legal notes
=================
| SPDX-FileCopyrightText: © 2022 ekvip automation GmbH <info@ekvip.de>
| SPDX-License-Identifier: Apache-2.0
| For details check: Apache-2.0_

.. _Apache-2.0: https://www.apache.org/licenses/LICENSE-2.0

.. _Apache-2.THIS^.SIZE_ZERO: https://www.apache.org/licenses/LICENSE-2.THIS^.SIZE_ZERO

.. </legal notes>

*)

METHOD runMemoryAreaIsNotDynamicTests
VAR
	foo				:__XWORD;
	stackAddress	:PVOID;
END_VAR
RETURN (NOT TcUnit.TEST_ORDERED(THIS^.getTestNameFor('memoryAreaIsNotDynamic')));
stackAddress := ADR(foo);

THIS^.testMemoryAreaIsNotDynamic(
	address := THIS,
	sizeInBytes := THIS^.I_AM_FAT,
	symbol := 'THIS'
);
THIS^.testMemoryAreaIsNotDynamic(
	address := THIS^.NULL_POINTER,
	sizeInBytes := THIS^.SIZE_ZERO,
	symbol := 'THIS^.NULL_POINTER'
);
THIS^.testMemoryAreaIsNotDynamic(
	address := stackAddress,
	sizeInBytes := SIZEOF(__XWORD),
	symbol := 'stackAddress'
);
THIS^.testMemoryAreaIsNotDynamic(
	address := THIS^.oneByte,
	sizeInBytes := SIZEOF(BYTE),
	symbol := 'THIS^.oneByte'
);
THIS^.testMemoryAreaIsNotDynamic(
	address := THIS^.byteArray,
	sizeInBytes := THIS^.ARRAY_SIZE,
	symbol := 'THIS^.byteArray'
);
THIS^.testMemoryAreaIsNotDynamic(
	address := THIS^.cncAddress,
	sizeInBytes := THIS^.cncSize,
	symbol := 'THIS^.cncAddress'
);
THIS^.testMemoryAreaIsNotDynamic(
	address := THIS^.itsMeAgain,
	sizeInBytes := SIZEOF(PVOID),
	symbol := 'THIS^.itsMeAgain'
);
THIS^.testMemoryAreaIsNotDynamic(
	address := THIS^.itsMeAgain^,
	sizeInBytes := THIS^.I_AM_FAT,
	symbol := 'THIS^.itsMeAgain^'
);
THIS^.testMemoryAreaIsNotDynamic(
	address := THIS^.me,
	sizeInBytes := THIS^.I_AM_FAT,
	symbol := 'THIS^.me'
);
THIS^.testMemoryAreaIsNotDynamic(
	address := THIS^.myMom,
	sizeInBytes := SIZEOF(AbstractAssertorTest),
	symbol := 'THIS^.myMom'
);
THIS^.testMemoryAreaIsNotDynamic(
	address := THIS^.invalidByte,
	sizeInBytes := SIZEOF(BYTE),
	symbol := 'THIS^.invalidByte'
);

THIS^.testMemoryAreaIsNotDynamic(
	address := THIS^.itsMeAgain,
	sizeInBytes := THIS^.SIZE_ZERO,
	symbol := 'THIS^.itsMeAgain'
);
THIS^.testMemoryAreaIsNotDynamic(
	address := THIS,
	sizeInBytes := THIS^.SIZE_ZERO,
	symbol := 'THIS'
);
THIS^.testMemoryAreaIsNotDynamic(
	address := THIS^.NULL_POINTER,
	sizeInBytes := SIZEOF(PVOID),
	symbol := 'THIS^.NULL_POINTER'
);
THIS^.testMemoryAreaIsNotDynamic(
	address := stackAddress,
	sizeInBytes := THIS^.SIZE_ZERO,
	symbol := 'stackAddress'
);
THIS^.testMemoryAreaIsNotDynamic(
	address := THIS^.oneByte,
	sizeInBytes := THIS^.SIZE_ZERO,
	symbol := 'THIS^.oneByte'
);
THIS^.testMemoryAreaIsNotDynamic(
	address := THIS^.byteArray,
	sizeInBytes := THIS^.SIZE_ZERO,
	symbol := 'THIS^.byteArray'
);
THIS^.testMemoryAreaIsNotDynamic(
	address := THIS^.itsMeAgain,
	sizeInBytes := THIS^.SIZE_ZERO,
	symbol := 'THIS^.itsMeAgain'
);
THIS^.testMemoryAreaIsNotDynamic(
	address := THIS^.cncAddress,
	sizeInBytes := THIS^.SIZE_ZERO,
	symbol := 'THIS^.cncAddress'
);
THIS^.testMemoryAreaIsNotDynamic(
	address := THIS^.itsMeAgain^,
	sizeInBytes := THIS^.SIZE_ZERO,
	symbol := 'THIS^.itsMeAgain^'
);
THIS^.testMemoryAreaIsNotDynamic(
	address := THIS^.INVALID_POINTER,
	sizeInBytes := SIZEOF(PVOID),
	symbol := 'THIS^.INVALID_POINTER'
);
THIS^.testMemoryAreaIsNotDynamic(
	address := THIS^.myMom,
	sizeInBytes := THIS^.SIZE_ZERO,
	symbol := 'THIS^.myMom'
);
THIS^.testMemoryAreaIsNotDynamic(
	address := THIS^.invalidByte,
	sizeInBytes := THIS^.SIZE_ZERO,
	symbol := 'THIS^.invalidByte'
);

TcUnit.TEST_FINISHED();
END_METHOD

(*

short summary
==================
This test method tests ``assert.pointers.memoryAreaIsNotStatic``
method of CNM_AssertionInterfaceLib library with various inputs

.. <legal notes>

legal notes
=================
| SPDX-FileCopyrightText: © 2022 ekvip automation GmbH <info@ekvip.de>
| SPDX-License-Identifier: Apache-2.0
| For details check: Apache-2.0_

.. _Apache-2.0: https://www.apache.org/licenses/LICENSE-2.0

.. _Apache-2.THIS^.SIZE_ZERO: https://www.apache.org/licenses/LICENSE-2.THIS^.SIZE_ZERO

.. </legal notes>

*)

METHOD runMemoryAreaIsNotStaticTests
VAR
	foo				:__XWORD;
	stackAddress	:PVOID;
END_VAR
RETURN (NOT TcUnit.TEST_ORDERED(THIS^.getTestNameFor('memoryAreaIsNotStatic')));
stackAddress := ADR(foo);

THIS^.testMemoryAreaIsNotStatic(
	address := THIS,
	sizeInBytes := THIS^.I_AM_FAT,
	symbol := 'THIS'
);
THIS^.testMemoryAreaIsNotStatic(
	address := THIS^.NULL_POINTER,
	sizeInBytes := THIS^.SIZE_ZERO,
	symbol := 'THIS^.NULL_POINTER'
);
THIS^.testMemoryAreaIsNotStatic(
	address := stackAddress,
	sizeInBytes := SIZEOF(__XWORD),
	symbol := 'stackAddress'
);
THIS^.testMemoryAreaIsNotStatic(
	address := THIS^.oneByte,
	sizeInBytes := SIZEOF(BYTE),
	symbol := 'THIS^.oneByte'
);
THIS^.testMemoryAreaIsNotStatic(
	address := THIS^.byteArray,
	sizeInBytes := THIS^.ARRAY_SIZE,
	symbol := 'THIS^.byteArray'
);
THIS^.testMemoryAreaIsNotStatic(
	address := THIS^.cncAddress,
	sizeInBytes := THIS^.cncSize,
	symbol := 'THIS^.cncAddress'
);
THIS^.testMemoryAreaIsNotStatic(
	address := THIS^.itsMeAgain,
	sizeInBytes := SIZEOF(PVOID),
	symbol := 'THIS^.itsMeAgain'
);
THIS^.testMemoryAreaIsNotStatic(
	address := THIS^.itsMeAgain^,
	sizeInBytes := THIS^.I_AM_FAT,
	symbol := 'THIS^.itsMeAgain^'
);
THIS^.testMemoryAreaIsNotStatic(
	address := THIS^.me,
	sizeInBytes := THIS^.I_AM_FAT,
	symbol := 'THIS^.me'
);
THIS^.testMemoryAreaIsNotStatic(
	address := THIS^.myMom,
	sizeInBytes := SIZEOF(AbstractAssertorTest),
	symbol := 'THIS^.myMom'
);
THIS^.testMemoryAreaIsNotStatic(
	address := THIS^.invalidByte,
	sizeInBytes := SIZEOF(BYTE),
	symbol := 'THIS^.invalidByte'
);

THIS^.testMemoryAreaIsNotStatic(
	address := THIS^.itsMeAgain,
	sizeInBytes := THIS^.SIZE_ZERO,
	symbol := 'THIS^.itsMeAgain'
);
THIS^.testMemoryAreaIsNotStatic(
	address := THIS,
	sizeInBytes := THIS^.SIZE_ZERO,
	symbol := 'THIS'
);
THIS^.testMemoryAreaIsNotStatic(
	address := THIS^.NULL_POINTER,
	sizeInBytes := SIZEOF(PVOID),
	symbol := 'THIS^.NULL_POINTER'
);
THIS^.testMemoryAreaIsNotStatic(
	address := stackAddress,
	sizeInBytes := THIS^.SIZE_ZERO,
	symbol := 'stackAddress'
);
THIS^.testMemoryAreaIsNotStatic(
	address := THIS^.oneByte,
	sizeInBytes := THIS^.SIZE_ZERO,
	symbol := 'THIS^.oneByte'
);
THIS^.testMemoryAreaIsNotStatic(
	address := THIS^.byteArray,
	sizeInBytes := THIS^.SIZE_ZERO,
	symbol := 'THIS^.byteArray'
);
THIS^.testMemoryAreaIsNotStatic(
	address := THIS^.itsMeAgain,
	sizeInBytes := THIS^.SIZE_ZERO,
	symbol := 'THIS^.itsMeAgain'
);
THIS^.testMemoryAreaIsNotStatic(
	address := THIS^.cncAddress,
	sizeInBytes := THIS^.SIZE_ZERO,
	symbol := 'THIS^.cncAddress'
);
THIS^.testMemoryAreaIsNotStatic(
	address := THIS^.itsMeAgain^,
	sizeInBytes := THIS^.SIZE_ZERO,
	symbol := 'THIS^.itsMeAgain^'
);
THIS^.testMemoryAreaIsNotStatic(
	address := THIS^.INVALID_POINTER,
	sizeInBytes := SIZEOF(PVOID),
	symbol := 'THIS^.INVALID_POINTER'
);
THIS^.testMemoryAreaIsNotStatic(
	address := THIS^.myMom,
	sizeInBytes := THIS^.SIZE_ZERO,
	symbol := 'THIS^.myMom'
);
THIS^.testMemoryAreaIsNotStatic(
	address := THIS^.invalidByte,
	sizeInBytes := THIS^.SIZE_ZERO,
	symbol := 'THIS^.invalidByte'
);

TcUnit.TEST_FINISHED();
END_METHOD

(*

short summary
==================
This test method tests ``assert.pointers.memoryAreaIsNotUnkown``
method of CNM_AssertionInterfaceLib library with various inputs

.. <legal notes>

legal notes
=================
| SPDX-FileCopyrightText: © 2022 ekvip automation GmbH <info@ekvip.de>
| SPDX-License-Identifier: Apache-2.0
| For details check: Apache-2.0_

.. _Apache-2.0: https://www.apache.org/licenses/LICENSE-2.0

.. _Apache-2.THIS^.SIZE_ZERO: https://www.apache.org/licenses/LICENSE-2.THIS^.SIZE_ZERO

.. </legal notes>

*)

METHOD runMemoryAreaIsNotUnknownTests
VAR
	foo				:__XWORD;
	stackAddress	:PVOID;
END_VAR
RETURN (NOT TcUnit.TEST_ORDERED(THIS^.getTestNameFor('memoryAreaIsNotUnkown')));
stackAddress := ADR(foo);

THIS^.testMemoryAreaIsNotUnknown(
	address := THIS,
	sizeInBytes := THIS^.I_AM_FAT,
	symbol := 'THIS'
);
THIS^.testMemoryAreaIsNotUnknown(
	address := THIS^.NULL_POINTER,
	sizeInBytes := THIS^.SIZE_ZERO,
	symbol := 'THIS^.NULL_POINTER'
);
THIS^.testMemoryAreaIsNotUnknown(
	address := stackAddress,
	sizeInBytes := SIZEOF(__XWORD),
	symbol := 'stackAddress'
);
THIS^.testMemoryAreaIsNotUnknown(
	address := THIS^.oneByte,
	sizeInBytes := SIZEOF(BYTE),
	symbol := 'THIS^.oneByte'
);
THIS^.testMemoryAreaIsNotUnknown(
	address := THIS^.byteArray,
	sizeInBytes := THIS^.ARRAY_SIZE,
	symbol := 'THIS^.byteArray'
);
THIS^.testMemoryAreaIsNotUnknown(
	address := THIS^.cncAddress,
	sizeInBytes := THIS^.cncSize,
	symbol := 'THIS^.cncAddress'
);
THIS^.testMemoryAreaIsNotUnknown(
	address := THIS^.itsMeAgain,
	sizeInBytes := SIZEOF(PVOID),
	symbol := 'THIS^.itsMeAgain'
);
THIS^.testMemoryAreaIsNotUnknown(
	address := THIS^.itsMeAgain^,
	sizeInBytes := THIS^.I_AM_FAT,
	symbol := 'THIS^.itsMeAgain^'
);
THIS^.testMemoryAreaIsNotUnknown(
	address := THIS^.me,
	sizeInBytes := THIS^.I_AM_FAT,
	symbol := 'THIS^.me'
);
THIS^.testMemoryAreaIsNotUnknown(
	address := THIS^.myMom,
	sizeInBytes := SIZEOF(AbstractAssertorTest),
	symbol := 'THIS^.myMom'
);
THIS^.testMemoryAreaIsNotUnknown(
	address := THIS^.invalidByte,
	sizeInBytes := SIZEOF(BYTE),
	symbol := 'THIS^.invalidByte'
);

THIS^.testMemoryAreaIsNotUnknown(
	address := THIS^.itsMeAgain,
	sizeInBytes := THIS^.SIZE_ZERO,
	symbol := 'THIS^.itsMeAgain'
);
THIS^.testMemoryAreaIsNotUnknown(
	address := THIS,
	sizeInBytes := THIS^.SIZE_ZERO,
	symbol := 'THIS'
);
THIS^.testMemoryAreaIsNotUnknown(
	address := THIS^.NULL_POINTER,
	sizeInBytes := SIZEOF(PVOID),
	symbol := 'THIS^.NULL_POINTER'
);
THIS^.testMemoryAreaIsNotUnknown(
	address := stackAddress,
	sizeInBytes := THIS^.SIZE_ZERO,
	symbol := 'stackAddress'
);
THIS^.testMemoryAreaIsNotUnknown(
	address := THIS^.oneByte,
	sizeInBytes := THIS^.SIZE_ZERO,
	symbol := 'THIS^.oneByte'
);
THIS^.testMemoryAreaIsNotUnknown(
	address := THIS^.byteArray,
	sizeInBytes := THIS^.SIZE_ZERO,
	symbol := 'THIS^.byteArray'
);
THIS^.testMemoryAreaIsNotUnknown(
	address := THIS^.itsMeAgain,
	sizeInBytes := THIS^.SIZE_ZERO,
	symbol := 'THIS^.itsMeAgain'
);
THIS^.testMemoryAreaIsNotUnknown(
	address := THIS^.cncAddress,
	sizeInBytes := THIS^.SIZE_ZERO,
	symbol := 'THIS^.cncAddress'
);
THIS^.testMemoryAreaIsNotUnknown(
	address := THIS^.itsMeAgain^,
	sizeInBytes := THIS^.SIZE_ZERO,
	symbol := 'THIS^.itsMeAgain^'
);
THIS^.testMemoryAreaIsNotUnknown(
	address := THIS^.INVALID_POINTER,
	sizeInBytes := SIZEOF(PVOID),
	symbol := 'THIS^.INVALID_POINTER'
);
THIS^.testMemoryAreaIsNotUnknown(
	address := THIS^.myMom,
	sizeInBytes := THIS^.SIZE_ZERO,
	symbol := 'THIS^.myMom'
);
THIS^.testMemoryAreaIsNotUnknown(
	address := THIS^.invalidByte,
	sizeInBytes := THIS^.SIZE_ZERO,
	symbol := 'THIS^.invalidByte'
);

TcUnit.TEST_FINISHED();
END_METHOD

(*

short summary
==================
This test method tests ``assert.pointers.memoryAreaIsStatic``
method of CNM_AssertionInterfaceLib library with various inputs

.. <legal notes>

legal notes
=================
| SPDX-FileCopyrightText: © 2022 ekvip automation GmbH <info@ekvip.de>
| SPDX-License-Identifier: Apache-2.0
| For details check: Apache-2.0_

.. _Apache-2.0: https://www.apache.org/licenses/LICENSE-2.0

.. _Apache-2.THIS^.SIZE_ZERO: https://www.apache.org/licenses/LICENSE-2.THIS^.SIZE_ZERO

.. </legal notes>

*)

METHOD runMemoryAreaIsStaticTests
VAR
	foo				:__XWORD;
	stackAddress	:PVOID;
END_VAR
RETURN (NOT TcUnit.TEST_ORDERED(THIS^.getTestNameFor('memoryAreaIsStatic')));
stackAddress := ADR(foo);

THIS^.testMemoryAreaIsStatic(
	address := THIS,
	sizeInBytes := THIS^.I_AM_FAT,
	symbol := 'THIS'
);
THIS^.testMemoryAreaIsStatic(
	address := THIS^.NULL_POINTER,
	sizeInBytes := THIS^.SIZE_ZERO,
	symbol := 'THIS^.NULL_POINTER'
);
THIS^.testMemoryAreaIsStatic(
	address := stackAddress,
	sizeInBytes := SIZEOF(__XWORD),
	symbol := 'stackAddress'
);
THIS^.testMemoryAreaIsStatic(
	address := THIS^.oneByte,
	sizeInBytes := SIZEOF(BYTE),
	symbol := 'THIS^.oneByte'
);
THIS^.testMemoryAreaIsStatic(
	address := THIS^.byteArray,
	sizeInBytes := THIS^.ARRAY_SIZE,
	symbol := 'THIS^.byteArray'
);
THIS^.testMemoryAreaIsStatic(
	address := THIS^.cncAddress,
	sizeInBytes := THIS^.cncSize,
	symbol := 'THIS^.cncAddress'
);
THIS^.testMemoryAreaIsStatic(
	address := THIS^.itsMeAgain,
	sizeInBytes := SIZEOF(PVOID),
	symbol := 'THIS^.itsMeAgain'
);
THIS^.testMemoryAreaIsStatic(
	address := THIS^.itsMeAgain^,
	sizeInBytes := THIS^.I_AM_FAT,
	symbol := 'THIS^.itsMeAgain^'
);
THIS^.testMemoryAreaIsStatic(
	address := THIS^.me,
	sizeInBytes := THIS^.I_AM_FAT,
	symbol := 'THIS^.me'
);
THIS^.testMemoryAreaIsStatic(
	address := THIS^.myMom,
	sizeInBytes := SIZEOF(AbstractAssertorTest),
	symbol := 'THIS^.myMom'
);
THIS^.testMemoryAreaIsStatic(
	address := THIS^.invalidByte,
	sizeInBytes := SIZEOF(BYTE),
	symbol := 'THIS^.invalidByte'
);

THIS^.testMemoryAreaIsStatic(
	address := THIS^.itsMeAgain,
	sizeInBytes := THIS^.SIZE_ZERO,
	symbol := 'THIS^.itsMeAgain'
);
THIS^.testMemoryAreaIsStatic(
	address := THIS,
	sizeInBytes := THIS^.SIZE_ZERO,
	symbol := 'THIS'
);
THIS^.testMemoryAreaIsStatic(
	address := THIS^.NULL_POINTER,
	sizeInBytes := SIZEOF(PVOID),
	symbol := 'THIS^.NULL_POINTER'
);
THIS^.testMemoryAreaIsStatic(
	address := stackAddress,
	sizeInBytes := THIS^.SIZE_ZERO,
	symbol := 'stackAddress'
);
THIS^.testMemoryAreaIsStatic(
	address := THIS^.oneByte,
	sizeInBytes := THIS^.SIZE_ZERO,
	symbol := 'THIS^.oneByte'
);
THIS^.testMemoryAreaIsStatic(
	address := THIS^.byteArray,
	sizeInBytes := THIS^.SIZE_ZERO,
	symbol := 'THIS^.byteArray'
);
THIS^.testMemoryAreaIsStatic(
	address := THIS^.itsMeAgain,
	sizeInBytes := THIS^.SIZE_ZERO,
	symbol := 'THIS^.itsMeAgain'
);
THIS^.testMemoryAreaIsStatic(
	address := THIS^.cncAddress,
	sizeInBytes := THIS^.SIZE_ZERO,
	symbol := 'THIS^.cncAddress'
);
THIS^.testMemoryAreaIsStatic(
	address := THIS^.itsMeAgain^,
	sizeInBytes := THIS^.SIZE_ZERO,
	symbol := 'THIS^.itsMeAgain^'
);
THIS^.testMemoryAreaIsStatic(
	address := THIS^.INVALID_POINTER,
	sizeInBytes := SIZEOF(PVOID),
	symbol := 'THIS^.INVALID_POINTER'
);
THIS^.testMemoryAreaIsStatic(
	address := THIS^.myMom,
	sizeInBytes := THIS^.SIZE_ZERO,
	symbol := 'THIS^.myMom'
);
THIS^.testMemoryAreaIsStatic(
	address := THIS^.invalidByte,
	sizeInBytes := THIS^.SIZE_ZERO,
	symbol := 'THIS^.invalidByte'
);

TcUnit.TEST_FINISHED();
END_METHOD

(*

short summary
==================
This test method tests ``assert.pointers.memoryAreaIsUnkown``
method of CNM_AssertionInterfaceLib library with various inputs

.. <legal notes>

legal notes
=================
| SPDX-FileCopyrightText: © 2022 ekvip automation GmbH <info@ekvip.de>
| SPDX-License-Identifier: Apache-2.0
| For details check: Apache-2.0_

.. _Apache-2.0: https://www.apache.org/licenses/LICENSE-2.0

.. _Apache-2.THIS^.SIZE_ZERO: https://www.apache.org/licenses/LICENSE-2.THIS^.SIZE_ZERO

.. </legal notes>

*)

METHOD runMemoryAreaIsUnknownTests
VAR
	foo				:__XWORD;
	stackAddress	:PVOID;
END_VAR
RETURN (NOT TcUnit.TEST_ORDERED(THIS^.getTestNameFor('memoryAreaIsUnkown')));
stackAddress := ADR(foo);

THIS^.testMemoryAreaIsUnknown(
	address := THIS,
	sizeInBytes := THIS^.I_AM_FAT,
	symbol := 'THIS'
);
THIS^.testMemoryAreaIsUnknown(
	address := THIS^.NULL_POINTER,
	sizeInBytes := THIS^.SIZE_ZERO,
	symbol := 'THIS^.NULL_POINTER'
);
THIS^.testMemoryAreaIsUnknown(
	address := stackAddress,
	sizeInBytes := SIZEOF(__XWORD),
	symbol := 'stackAddress'
);
THIS^.testMemoryAreaIsUnknown(
	address := THIS^.oneByte,
	sizeInBytes := SIZEOF(BYTE),
	symbol := 'THIS^.oneByte'
);
THIS^.testMemoryAreaIsUnknown(
	address := THIS^.byteArray,
	sizeInBytes := THIS^.ARRAY_SIZE,
	symbol := 'THIS^.byteArray'
);
THIS^.testMemoryAreaIsUnknown(
	address := THIS^.cncAddress,
	sizeInBytes := THIS^.cncSize,
	symbol := 'THIS^.cncAddress'
);
THIS^.testMemoryAreaIsUnknown(
	address := THIS^.itsMeAgain,
	sizeInBytes := SIZEOF(PVOID),
	symbol := 'THIS^.itsMeAgain'
);
THIS^.testMemoryAreaIsUnknown(
	address := THIS^.itsMeAgain^,
	sizeInBytes := THIS^.I_AM_FAT,
	symbol := 'THIS^.itsMeAgain^'
);
THIS^.testMemoryAreaIsUnknown(
	address := THIS^.me,
	sizeInBytes := THIS^.I_AM_FAT,
	symbol := 'THIS^.me'
);
THIS^.testMemoryAreaIsUnknown(
	address := THIS^.myMom,
	sizeInBytes := SIZEOF(AbstractAssertorTest),
	symbol := 'THIS^.myMom'
);
THIS^.testMemoryAreaIsUnknown(
	address := THIS^.invalidByte,
	sizeInBytes := SIZEOF(BYTE),
	symbol := 'THIS^.invalidByte'
);

THIS^.testMemoryAreaIsUnknown(
	address := THIS^.itsMeAgain,
	sizeInBytes := THIS^.SIZE_ZERO,
	symbol := 'THIS^.itsMeAgain'
);
THIS^.testMemoryAreaIsUnknown(
	address := THIS,
	sizeInBytes := THIS^.SIZE_ZERO,
	symbol := 'THIS'
);
THIS^.testMemoryAreaIsUnknown(
	address := THIS^.NULL_POINTER,
	sizeInBytes := SIZEOF(PVOID),
	symbol := 'THIS^.NULL_POINTER'
);
THIS^.testMemoryAreaIsUnknown(
	address := stackAddress,
	sizeInBytes := THIS^.SIZE_ZERO,
	symbol := 'stackAddress'
);
THIS^.testMemoryAreaIsUnknown(
	address := THIS^.oneByte,
	sizeInBytes := THIS^.SIZE_ZERO,
	symbol := 'THIS^.oneByte'
);
THIS^.testMemoryAreaIsUnknown(
	address := THIS^.byteArray,
	sizeInBytes := THIS^.SIZE_ZERO,
	symbol := 'THIS^.byteArray'
);
THIS^.testMemoryAreaIsUnknown(
	address := THIS^.itsMeAgain,
	sizeInBytes := THIS^.SIZE_ZERO,
	symbol := 'THIS^.itsMeAgain'
);
THIS^.testMemoryAreaIsUnknown(
	address := THIS^.cncAddress,
	sizeInBytes := THIS^.SIZE_ZERO,
	symbol := 'THIS^.cncAddress'
);
THIS^.testMemoryAreaIsUnknown(
	address := THIS^.itsMeAgain^,
	sizeInBytes := THIS^.SIZE_ZERO,
	symbol := 'THIS^.itsMeAgain^'
);
THIS^.testMemoryAreaIsUnknown(
	address := THIS^.INVALID_POINTER,
	sizeInBytes := SIZEOF(PVOID),
	symbol := 'THIS^.INVALID_POINTER'
);
THIS^.testMemoryAreaIsUnknown(
	address := THIS^.myMom,
	sizeInBytes := THIS^.SIZE_ZERO,
	symbol := 'THIS^.myMom'
);
THIS^.testMemoryAreaIsUnknown(
	address := THIS^.invalidByte,
	sizeInBytes := THIS^.SIZE_ZERO,
	symbol := 'THIS^.invalidByte'
);

TcUnit.TEST_FINISHED();
END_METHOD

(*

short summary
==================
This test method tests ``assert.pointers.isEqualTo``
method of CNM_AssertionInterfaceLib library, 
it provides the possibility to handover test data via parameter 


.. <legal notes>

legal notes
=================
| SPDX-FileCopyrightText: © 2022 ekvip automation GmbH <info@ekvip.de>
| SPDX-License-Identifier: Apache-2.0
| For details check: Apache-2.0_

.. _Apache-2.0: https://www.apache.org/licenses/LICENSE-2.0

.. </legal notes>

parameters
==========

*)

METHOD testIsEqualTo
VAR_INPUT
	(* for the test it's the parameter ``address1`` *)
	address1	:PVOID;
	(* for the test it's the parameter ``address2`` *)
	address2	:PVOID;
END_VAR
VAR
	(* just the expectation if the assertion to test must be worng or true *)
	assertionIsWrong		:BOOL;
	(* contains the format string for the test message *)
	message					:Tc2_System.T_MaxString;
	(* TwinCAT printf with the test message *)
	messageStringBuilder	:Tc2_Utilities.FB_FormatString;
END_VAR
THIS^.assertorContainer.resetAssertor();

assertionIsWrong := (address1 <> address2);
message := SEL(
	assertionIsWrong,
	'address1 is 16#%X address2 is 16#%X assertion must be TRUE', 
	'address1 is 16#%X address2 is 16#%X assertion must be FALSE'
);
messageStringBuilder(
	sFormat := message,
	arg1 := THIS^.AnyToArg(address1),
	arg2 := THIS^.AnyToArg(address2)
);

THIS^.assertorContainer.assertor.assert.pointers.isEqualTo(
	address1 := address1,
	address2 := address2,
	message := ''
);

THIS^.AssertEquals_BOOL(
	Expected 	:= assertionIsWrong,
	Actual 		:= THIS^.assertorContainer.wasAssertionWrong,
	Message 	:= messageStringBuilder.sOut
);
END_METHOD

(*

short summary
==================
This test method tests ``assert.pointers.isNotNull``
method of CNM_AssertionInterfaceLib library, 
it provides the possibility to handover test data via parameter 


.. <legal notes>

legal notes
=================
| SPDX-FileCopyrightText: © 2022 ekvip automation GmbH <info@ekvip.de>
| SPDX-License-Identifier: Apache-2.0
| For details check: Apache-2.0_

.. _Apache-2.0: https://www.apache.org/licenses/LICENSE-2.0

.. </legal notes>

parameters
==========

*)

METHOD testIsNotNull
VAR_INPUT
	(* for the test it's the parameter ``address`` *)
	address		:PVOID;
	(* just the name of the pointer *)
	symbol		:Tc2_System.T_MaxString;
END_VAR
VAR
	(* just the expectation if the assertion to test must be worng or true *)
	assertionIsWrong		:BOOL;
	(* contains the format string for the test message *)
	message					:Tc2_System.T_MaxString;
	(* TwinCAT printf with the test message *)
	messageStringBuilder	:Tc2_Utilities.FB_FormatString;
END_VAR
THIS^.assertorContainer.resetAssertor();

assertionIsWrong := (address = THIS^.NULL_POINTER);
message := SEL(
	assertionIsWrong,
	'address is 16#%X ($'%s$') assertion must be TRUE', 
	'address is 16#%X ($'%s$') assertion must be FALSE'
);
messageStringBuilder(
	sFormat := message,
	arg1 := THIS^.AnyToArg(address),
	arg2 := THIS^.AnyToArg(symbol)
);

THIS^.assertorContainer.assertor.assert.pointers.isNotNull(
	address := address,
	message := ''
);

THIS^.AssertEquals_BOOL(
	Expected 	:= assertionIsWrong,
	Actual 		:= THIS^.assertorContainer.wasAssertionWrong,
	Message 	:= messageStringBuilder.sOut
);
END_METHOD

(*

short summary
==================
This test method tests ``assert.pointers.isNull``
method of CNM_AssertionInterfaceLib library, 
it provides the possibility to handover test data via parameter 


.. <legal notes>

legal notes
=================
| SPDX-FileCopyrightText: © 2022 ekvip automation GmbH <info@ekvip.de>
| SPDX-License-Identifier: Apache-2.0
| For details check: Apache-2.0_

.. _Apache-2.0: https://www.apache.org/licenses/LICENSE-2.0

.. </legal notes>

parameters
==========

*)

METHOD testIsNull
VAR_INPUT
	(* for the test it's the parameter ``address`` *)
	address		:PVOID;
	(* just the name of the pointer *)
	symbol		:Tc2_System.T_MaxString;
END_VAR
VAR
	(* just the expectation if the assertion to test must be worng or true *)
	assertionIsWrong		:BOOL;
	(* contains the format string for the test message *)
	message					:Tc2_System.T_MaxString;
	(* TwinCAT printf with the test message *)
	messageStringBuilder	:Tc2_Utilities.FB_FormatString;
END_VAR
THIS^.assertorContainer.resetAssertor();

assertionIsWrong := (address <> THIS^.NULL_POINTER);
message := SEL(
	assertionIsWrong,
	'address is 16#%X ($'%s$') assertion must be TRUE', 
	'address is 16#%X ($'%s$') assertion must be FALSE'
);
messageStringBuilder(
	sFormat := message,
	arg1 := THIS^.AnyToArg(address),
	arg2 := THIS^.AnyToArg(symbol)
);

THIS^.assertorContainer.assertor.assert.pointers.isNull(
	address := address,
	message := ''
);

THIS^.AssertEquals_BOOL(
	Expected 	:= assertionIsWrong,
	Actual 		:= THIS^.assertorContainer.wasAssertionWrong,
	Message 	:= messageStringBuilder.sOut
);
END_METHOD

(*

short summary
==================
This test method tests ``assert.pointers.isValid``
method of CNM_AssertionInterfaceLib library, 
it provides the possibility to handover test data via parameter 

.. <legal notes>

legal notes
=================
| SPDX-FileCopyrightText: © 2022 ekvip automation GmbH <info@ekvip.de>
| SPDX-License-Identifier: Apache-2.0
| For details check: Apache-2.0_

.. _Apache-2.0: https://www.apache.org/licenses/LICENSE-2.0

.. </legal notes>

parameters
==========

*)

METHOD testIsValid
VAR_INPUT
	(* for the test it's the parameter ``address`` *)
	address		:PVOID;
	(* for the test it's the parameter ``sizeInBytes`` *)
	sizeInBytes	:UDINT;
	(* just the name of the pointer *)
	symbol		:Tc2_System.T_MaxString;
END_VAR
VAR
	(* just the expectation if the assertion to test must be worng or true *)
	assertionIsWrong		:BOOL;
	(* contains the format string for the test message *)
	message					:Tc2_System.T_MaxString;
	(* TwinCAT printf with the test message *)
	messageStringBuilder	:Tc2_Utilities.FB_FormatString;
	(* return value of Tc2_System.F_CheckMemoryArea *)
	memoryArea				:Tc2_System.E_TcMemoryArea;
	(*  return value of Tc2_System.F_CheckMemoryArea as string *)
	areaString				:Tc2_System.T_MaxString;
	{IF hasvalue (RegisterSize, '32')}
	(* lets try if it's possible to read something from the address *)
	validityTester			:POINTER TO BYTE;
	(* dummy variable with the value *)
	value					:BYTE;
	(* exception code *)
	e						:ExceptionCode;
	(* just to test it over all elemets *)
	count					:UDINT;
	{END_IF}
END_VAR
THIS^.assertorContainer.resetAssertor();

memoryArea	:= Tc2_System.F_CheckMemoryArea(address, sizeInBytes);
areaString	:= THIS^.memoryAreaToString(memoryArea);

{IF hasvalue (RegisterSize, '32')}
validityTester := address;
assertionIsWrong := (
	(sizeInBytes <= THIS^.SIZE_ZERO)
	AND (address > THIS^.NULL_POINTER)
);
__TRY
	IF (NOT assertionIsWrong) THEN
		FOR byteCount := 0 TO (sizeInBytes-1) DO
			value := validityTester[byteCount];
		END_FOR
	END_IF
__CATCH(e)
	assertionIsWrong := TRUE;
__ENDTRY
{ELSE}
assertionIsWrong := (
	(memoryArea = Tc2_System.E_TcMemoryArea.Unknown)
	OR (sizeInBytes <= THIS^.SIZE_ZERO)
);
{END_IF}

message := SEL(
	assertionIsWrong,
	'address is 16#%X ($'%s$') sizeInBytes is %d return value of Tc2_System.F_CheckMemoryArea is $'%s$' assertion must be TRUE', 
	'address is 16#%X ($'%s$') sizeInBytes is %d return value of Tc2_System.F_CheckMemoryArea is $'%s$' assertion must be FALSE'
);
messageStringBuilder(
	sFormat := message,
	arg1 := THIS^.AnyToArg(address),
	arg2 := THIS^.AnyToArg(symbol),
	arg3 := THIS^.AnyToArg(sizeInBytes),
	arg4 := THIS^.AnyToArg(areaString)
);

THIS^.assertorContainer.assertor.assert.pointers.isValid(
	address := address,
	sizeInBytes := sizeInBytes,
	message := ''
);

THIS^.AssertEquals_BOOL(
	Expected 	:= assertionIsWrong,
	Actual 		:= THIS^.assertorContainer.wasAssertionWrong,
	Message 	:= messageStringBuilder.sOut
);
END_METHOD

(*

short summary
==================
This test method tests ``assert.pointers.memoryAreaIsCnc``
method of CNM_AssertionInterfaceLib library, 
it provides the possibility to handover test data via parameter 

.. <legal notes>

legal notes
=================
| SPDX-FileCopyrightText: © 2022 ekvip automation GmbH <info@ekvip.de>
| SPDX-License-Identifier: Apache-2.0
| For details check: Apache-2.0_

.. _Apache-2.0: https://www.apache.org/licenses/LICENSE-2.0

.. </legal notes>

parameters
==========

*)

METHOD testMemoryAreaIsCnc
VAR_INPUT
	(* for the test it's the parameter ``address`` *)
	address		:PVOID;
	(* for the test it's the parameter ``sizeInBytes`` *)
	sizeInBytes	:UDINT;
	(* just the name of the pointer *)
	symbol		:Tc2_System.T_MaxString;
END_VAR
VAR
	(* just the expectation if the assertion to test must be worng or true *)
	assertionIsWrong		:BOOL;
	(* contains the format string for the test message *)
	message					:Tc2_System.T_MaxString;
	(* TwinCAT printf with the test message *)
	messageStringBuilder	:Tc2_Utilities.FB_FormatString;
	(* return value of Tc2_System.F_CheckMemoryArea *)
	memoryArea				:Tc2_System.E_TcMemoryArea;
	(*  return value of Tc2_System.F_CheckMemoryArea as string *)
	areaString				:Tc2_System.T_MaxString;
END_VAR
THIS^.assertorContainer.resetAssertor();

memoryArea	:= Tc2_System.F_CheckMemoryArea(address, sizeInBytes);
areaString	:= THIS^.memoryAreaToString(memoryArea);
assertionIsWrong := (memoryArea <> Tc2_System.E_TcMemoryArea.CNC);

message := SEL(
	assertionIsWrong,
	'address is 16#%X ($'%s$') sizeInBytes is %d return value of Tc2_System.F_CheckMemoryArea is $'%s$' assertion must be TRUE', 
	'address is 16#%X ($'%s$') sizeInBytes is %d return value of Tc2_System.F_CheckMemoryArea is $'%s$' assertion must be FALSE'
);
messageStringBuilder(
	sFormat := message,
	arg1 := THIS^.AnyToArg(address),
	arg2 := THIS^.AnyToArg(symbol),
	arg3 := THIS^.AnyToArg(sizeInBytes),
	arg4 := THIS^.AnyToArg(areaString)
);

THIS^.assertorContainer.assertor.assert.pointers.memoryAreaIsCnc(
	address := address,
	sizeInBytes := sizeInBytes,
	message := ''
);

THIS^.AssertEquals_BOOL(
	Expected 	:= assertionIsWrong,
	Actual 		:= THIS^.assertorContainer.wasAssertionWrong,
	Message 	:= messageStringBuilder.sOut
);
END_METHOD

(*

short summary
==================
This test method tests ``assert.pointers.memoryAreaIsDynamic``
method of CNM_AssertionInterfaceLib library, 
it provides the possibility to handover test data via parameter 

.. <legal notes>

legal notes
=================
| SPDX-FileCopyrightText: © 2022 ekvip automation GmbH <info@ekvip.de>
| SPDX-License-Identifier: Apache-2.0
| For details check: Apache-2.0_

.. _Apache-2.0: https://www.apache.org/licenses/LICENSE-2.0

.. </legal notes>

parameters
==========

*)

METHOD testMemoryAreaIsDynamic
VAR_INPUT
	(* for the test it's the parameter ``address`` *)
	address		:PVOID;
	(* for the test it's the parameter ``sizeInBytes`` *)
	sizeInBytes	:UDINT;
	(* just the name of the pointer *)
	symbol		:Tc2_System.T_MaxString;
END_VAR
VAR
	(* just the expectation if the assertion to test must be worng or true *)
	assertionIsWrong		:BOOL;
	(* contains the format string for the test message *)
	message					:Tc2_System.T_MaxString;
	(* TwinCAT printf with the test message *)
	messageStringBuilder	:Tc2_Utilities.FB_FormatString;
	(* return value of Tc2_System.F_CheckMemoryArea *)
	memoryArea				:Tc2_System.E_TcMemoryArea;
	(*  return value of Tc2_System.F_CheckMemoryArea as string *)
	areaString				:Tc2_System.T_MaxString;
END_VAR
THIS^.assertorContainer.resetAssertor();

memoryArea	:= Tc2_System.F_CheckMemoryArea(address, sizeInBytes);
areaString	:= THIS^.memoryAreaToString(memoryArea);
assertionIsWrong := (memoryArea <> Tc2_System.E_TcMemoryArea.Dynamic);

message := SEL(
	assertionIsWrong,
	'address is 16#%X ($'%s$') sizeInBytes is %d return value of Tc2_System.F_CheckMemoryArea is $'%s$' assertion must be TRUE', 
	'address is 16#%X ($'%s$') sizeInBytes is %d return value of Tc2_System.F_CheckMemoryArea is $'%s$' assertion must be FALSE'
);
messageStringBuilder(
	sFormat := message,
	arg1 := THIS^.AnyToArg(address),
	arg2 := THIS^.AnyToArg(symbol),
	arg3 := THIS^.AnyToArg(sizeInBytes),
	arg4 := THIS^.AnyToArg(areaString)
);

THIS^.assertorContainer.assertor.assert.pointers.memoryAreaIsDynamic(
	address := address,
	sizeInBytes := sizeInBytes,
	message := ''
);

THIS^.AssertEquals_BOOL(
	Expected 	:= assertionIsWrong,
	Actual 		:= THIS^.assertorContainer.wasAssertionWrong,
	Message 	:= messageStringBuilder.sOut
);
END_METHOD

(*

short summary
==================
This test method tests ``assert.pointers.memoryAreaIsNotCnc``
method of CNM_AssertionInterfaceLib library, 
it provides the possibility to handover test data via parameter 

.. <legal notes>

legal notes
=================
| SPDX-FileCopyrightText: © 2022 ekvip automation GmbH <info@ekvip.de>
| SPDX-License-Identifier: Apache-2.0
| For details check: Apache-2.0_

.. _Apache-2.0: https://www.apache.org/licenses/LICENSE-2.0

.. </legal notes>

parameters
==========

*)

METHOD testMemoryAreaIsNotCnc
VAR_INPUT
	(* for the test it's the parameter ``address`` *)
	address		:PVOID;
	(* for the test it's the parameter ``sizeInBytes`` *)
	sizeInBytes	:UDINT;
	(* just the name of the pointer *)
	symbol		:Tc2_System.T_MaxString;
END_VAR
VAR
	(* just the expectation if the assertion to test must be worng or true *)
	assertionIsWrong		:BOOL;
	(* contains the format string for the test message *)
	message					:Tc2_System.T_MaxString;
	(* TwinCAT printf with the test message *)
	messageStringBuilder	:Tc2_Utilities.FB_FormatString;
	(* return value of Tc2_System.F_CheckMemoryArea *)
	memoryArea				:Tc2_System.E_TcMemoryArea;
	(*  return value of Tc2_System.F_CheckMemoryArea as string *)
	areaString				:Tc2_System.T_MaxString;
END_VAR
THIS^.assertorContainer.resetAssertor();

memoryArea	:= Tc2_System.F_CheckMemoryArea(address, sizeInBytes);
areaString	:= THIS^.memoryAreaToString(memoryArea);
assertionIsWrong := (memoryArea = Tc2_System.E_TcMemoryArea.CNC);

message := SEL(
	assertionIsWrong,
	'address is 16#%X ($'%s$') sizeInBytes is %d return value of Tc2_System.F_CheckMemoryArea is $'%s$' assertion must be TRUE', 
	'address is 16#%X ($'%s$') sizeInBytes is %d return value of Tc2_System.F_CheckMemoryArea is $'%s$' assertion must be FALSE'
);
messageStringBuilder(
	sFormat := message,
	arg1 := THIS^.AnyToArg(address),
	arg2 := THIS^.AnyToArg(symbol),
	arg3 := THIS^.AnyToArg(sizeInBytes),
	arg4 := THIS^.AnyToArg(areaString)
);

THIS^.assertorContainer.assertor.assert.pointers.memoryAreaIsNotCnc(
	address := address,
	sizeInBytes := sizeInBytes,
	message := ''
);

THIS^.AssertEquals_BOOL(
	Expected 	:= assertionIsWrong,
	Actual 		:= THIS^.assertorContainer.wasAssertionWrong,
	Message 	:= messageStringBuilder.sOut
);
END_METHOD

(*

short summary
==================
This test method tests ``assert.pointers.memoryAreaIsNotDynamic``
method of CNM_AssertionInterfaceLib library, 
it provides the possibility to handover test data via parameter 

.. <legal notes>

legal notes
=================
| SPDX-FileCopyrightText: © 2022 ekvip automation GmbH <info@ekvip.de>
| SPDX-License-Identifier: Apache-2.0
| For details check: Apache-2.0_

.. _Apache-2.0: https://www.apache.org/licenses/LICENSE-2.0

.. </legal notes>

parameters
==========

*)

METHOD testMemoryAreaIsNotDynamic
VAR_INPUT
	(* for the test it's the parameter ``address`` *)
	address		:PVOID;
	(* for the test it's the parameter ``sizeInBytes`` *)
	sizeInBytes	:UDINT;
	(* just the name of the pointer *)
	symbol		:Tc2_System.T_MaxString;
END_VAR
VAR
	(* just the expectation if the assertion to test must be worng or true *)
	assertionIsWrong		:BOOL;
	(* contains the format string for the test message *)
	message					:Tc2_System.T_MaxString;
	(* TwinCAT printf with the test message *)
	messageStringBuilder	:Tc2_Utilities.FB_FormatString;
	(* return value of Tc2_System.F_CheckMemoryArea *)
	memoryArea				:Tc2_System.E_TcMemoryArea;
	(*  return value of Tc2_System.F_CheckMemoryArea as string *)
	areaString				:Tc2_System.T_MaxString;
END_VAR
THIS^.assertorContainer.resetAssertor();

memoryArea	:= Tc2_System.F_CheckMemoryArea(address, sizeInBytes);
areaString	:= THIS^.memoryAreaToString(memoryArea);
assertionIsWrong := (memoryArea = Tc2_System.E_TcMemoryArea.Dynamic);

message := SEL(
	assertionIsWrong,
	'address is 16#%X ($'%s$') sizeInBytes is %d return value of Tc2_System.F_CheckMemoryArea is $'%s$' assertion must be TRUE', 
	'address is 16#%X ($'%s$') sizeInBytes is %d return value of Tc2_System.F_CheckMemoryArea is $'%s$' assertion must be FALSE'
);
messageStringBuilder(
	sFormat := message,
	arg1 := THIS^.AnyToArg(address),
	arg2 := THIS^.AnyToArg(symbol),
	arg3 := THIS^.AnyToArg(sizeInBytes),
	arg4 := THIS^.AnyToArg(areaString)
);

THIS^.assertorContainer.assertor.assert.pointers.memoryAreaIsNotDynamic(
	address := address,
	sizeInBytes := sizeInBytes,
	message := ''
);

THIS^.AssertEquals_BOOL(
	Expected 	:= assertionIsWrong,
	Actual 		:= THIS^.assertorContainer.wasAssertionWrong,
	Message 	:= messageStringBuilder.sOut
);
END_METHOD

(*

short summary
==================
This test method tests ``assert.pointers.memoryAreaIsNotStatic``
method of CNM_AssertionInterfaceLib library, 
it provides the possibility to handover test data via parameter 

.. <legal notes>

legal notes
=================
| SPDX-FileCopyrightText: © 2022 ekvip automation GmbH <info@ekvip.de>
| SPDX-License-Identifier: Apache-2.0
| For details check: Apache-2.0_

.. _Apache-2.0: https://www.apache.org/licenses/LICENSE-2.0

.. </legal notes>

parameters
==========

*)

METHOD testMemoryAreaIsNotStatic
VAR_INPUT
	(* for the test it's the parameter ``address`` *)
	address		:PVOID;
	(* for the test it's the parameter ``sizeInBytes`` *)
	sizeInBytes	:UDINT;
	(* just the name of the pointer *)
	symbol		:Tc2_System.T_MaxString;
END_VAR
VAR
	(* just the expectation if the assertion to test must be worng or true *)
	assertionIsWrong		:BOOL;
	(* contains the format string for the test message *)
	message					:Tc2_System.T_MaxString;
	(* TwinCAT printf with the test message *)
	messageStringBuilder	:Tc2_Utilities.FB_FormatString;
	(* return value of Tc2_System.F_CheckMemoryArea *)
	memoryArea				:Tc2_System.E_TcMemoryArea;
	(*  return value of Tc2_System.F_CheckMemoryArea as string *)
	areaString				:Tc2_System.T_MaxString;
END_VAR
THIS^.assertorContainer.resetAssertor();

memoryArea	:= Tc2_System.F_CheckMemoryArea(address, sizeInBytes);
areaString	:= THIS^.memoryAreaToString(memoryArea);
assertionIsWrong := (memoryArea = Tc2_System.E_TcMemoryArea.Static);

message := SEL(
	assertionIsWrong,
	'address is 16#%X ($'%s$') sizeInBytes is %d return value of Tc2_System.F_CheckMemoryArea is $'%s$' assertion must be TRUE', 
	'address is 16#%X ($'%s$') sizeInBytes is %d return value of Tc2_System.F_CheckMemoryArea is $'%s$' assertion must be FALSE'
);
messageStringBuilder(
	sFormat := message,
	arg1 := THIS^.AnyToArg(address),
	arg2 := THIS^.AnyToArg(symbol),
	arg3 := THIS^.AnyToArg(sizeInBytes),
	arg4 := THIS^.AnyToArg(areaString)
);

THIS^.assertorContainer.assertor.assert.pointers.memoryAreaIsNotStatic(
	address := address,
	sizeInBytes := sizeInBytes,
	message := ''
);

THIS^.AssertEquals_BOOL(
	Expected 	:= assertionIsWrong,
	Actual 		:= THIS^.assertorContainer.wasAssertionWrong,
	Message 	:= messageStringBuilder.sOut
);
END_METHOD

(*

short summary
==================
This test method tests ``assert.pointers.memoryAreaIsNotUnkown``
method of CNM_AssertionInterfaceLib library, 
it provides the possibility to handover test data via parameter 

.. <legal notes>

legal notes
=================
| SPDX-FileCopyrightText: © 2022 ekvip automation GmbH <info@ekvip.de>
| SPDX-License-Identifier: Apache-2.0
| For details check: Apache-2.0_

.. _Apache-2.0: https://www.apache.org/licenses/LICENSE-2.0

.. </legal notes>

parameters
==========

*)

METHOD testMemoryAreaIsNotUnknown
VAR_INPUT
	(* for the test it's the parameter ``address`` *)
	address		:PVOID;
	(* for the test it's the parameter ``sizeInBytes`` *)
	sizeInBytes	:UDINT;
	(* just the name of the pointer *)
	symbol		:Tc2_System.T_MaxString;
END_VAR
VAR
	(* just the expectation if the assertion to test must be worng or true *)
	assertionIsWrong		:BOOL;
	(* contains the format string for the test message *)
	message					:Tc2_System.T_MaxString;
	(* TwinCAT printf with the test message *)
	messageStringBuilder	:Tc2_Utilities.FB_FormatString;
	(* return value of Tc2_System.F_CheckMemoryArea *)
	memoryArea				:Tc2_System.E_TcMemoryArea;
	(*  return value of Tc2_System.F_CheckMemoryArea as string *)
	areaString				:Tc2_System.T_MaxString;
END_VAR
THIS^.assertorContainer.resetAssertor();

memoryArea	:= Tc2_System.F_CheckMemoryArea(address, sizeInBytes);
areaString	:= THIS^.memoryAreaToString(memoryArea);
assertionIsWrong := (memoryArea = Tc2_System.E_TcMemoryArea.Unknown);

message := SEL(
	assertionIsWrong,
	'address is 16#%X ($'%s$') sizeInBytes is %d return value of Tc2_System.F_CheckMemoryArea is $'%s$' assertion must be TRUE', 
	'address is 16#%X ($'%s$') sizeInBytes is %d return value of Tc2_System.F_CheckMemoryArea is $'%s$' assertion must be FALSE'
);
messageStringBuilder(
	sFormat := message,
	arg1 := THIS^.AnyToArg(address),
	arg2 := THIS^.AnyToArg(symbol),
	arg3 := THIS^.AnyToArg(sizeInBytes),
	arg4 := THIS^.AnyToArg(areaString)
);

THIS^.assertorContainer.assertor.assert.pointers.memoryAreaIsNotUnkown(
	address := address,
	sizeInBytes := sizeInBytes,
	message := ''
);

THIS^.AssertEquals_BOOL(
	Expected 	:= assertionIsWrong,
	Actual 		:= THIS^.assertorContainer.wasAssertionWrong,
	Message 	:= messageStringBuilder.sOut
);
END_METHOD

(*

short summary
==================
This test method tests ``assert.pointers.memoryAreaIsStatic``
method of CNM_AssertionInterfaceLib library, 
it provides the possibility to handover test data via parameter 

.. <legal notes>

legal notes
=================
| SPDX-FileCopyrightText: © 2022 ekvip automation GmbH <info@ekvip.de>
| SPDX-License-Identifier: Apache-2.0
| For details check: Apache-2.0_

.. _Apache-2.0: https://www.apache.org/licenses/LICENSE-2.0

.. </legal notes>

parameters
==========

*)

METHOD testMemoryAreaIsStatic
VAR_INPUT
	(* for the test it's the parameter ``address`` *)
	address		:PVOID;
	(* for the test it's the parameter ``sizeInBytes`` *)
	sizeInBytes	:UDINT;
	(* just the name of the pointer *)
	symbol		:Tc2_System.T_MaxString;
END_VAR
VAR
	(* just the expectation if the assertion to test must be worng or true *)
	assertionIsWrong		:BOOL;
	(* contains the format string for the test message *)
	message					:Tc2_System.T_MaxString;
	(* TwinCAT printf with the test message *)
	messageStringBuilder	:Tc2_Utilities.FB_FormatString;
	(* return value of Tc2_System.F_CheckMemoryArea *)
	memoryArea				:Tc2_System.E_TcMemoryArea;
	(*  return value of Tc2_System.F_CheckMemoryArea as string *)
	areaString				:Tc2_System.T_MaxString;
END_VAR
THIS^.assertorContainer.resetAssertor();

memoryArea	:= Tc2_System.F_CheckMemoryArea(address, sizeInBytes);
areaString	:= THIS^.memoryAreaToString(memoryArea);
assertionIsWrong := (memoryArea <> Tc2_System.E_TcMemoryArea.Static);

message := SEL(
	assertionIsWrong,
	'address is 16#%X ($'%s$') sizeInBytes is %d return value of Tc2_System.F_CheckMemoryArea is $'%s$' assertion must be TRUE', 
	'address is 16#%X ($'%s$') sizeInBytes is %d return value of Tc2_System.F_CheckMemoryArea is $'%s$' assertion must be FALSE'
);
messageStringBuilder(
	sFormat := message,
	arg1 := THIS^.AnyToArg(address),
	arg2 := THIS^.AnyToArg(symbol),
	arg3 := THIS^.AnyToArg(sizeInBytes),
	arg4 := THIS^.AnyToArg(areaString)
);

THIS^.assertorContainer.assertor.assert.pointers.memoryAreaIsStatic(
	address := address,
	sizeInBytes := sizeInBytes,
	message := ''
);

THIS^.AssertEquals_BOOL(
	Expected 	:= assertionIsWrong,
	Actual 		:= THIS^.assertorContainer.wasAssertionWrong,
	Message 	:= messageStringBuilder.sOut
);
END_METHOD

(*

short summary
==================
This test method tests ``assert.pointers.memoryAreaIsUnkown``
method of CNM_AssertionInterfaceLib library, 
it provides the possibility to handover test data via parameter 

.. <legal notes>

legal notes
=================
| SPDX-FileCopyrightText: © 2022 ekvip automation GmbH <info@ekvip.de>
| SPDX-License-Identifier: Apache-2.0
| For details check: Apache-2.0_

.. _Apache-2.0: https://www.apache.org/licenses/LICENSE-2.0

.. </legal notes>

parameters
==========

*)

METHOD testMemoryAreaIsUnknown
VAR_INPUT
	(* for the test it's the parameter ``address`` *)
	address		:PVOID;
	(* for the test it's the parameter ``sizeInBytes`` *)
	sizeInBytes	:UDINT;
	(* just the name of the pointer *)
	symbol		:Tc2_System.T_MaxString;
END_VAR
VAR
	(* just the expectation if the assertion to test must be worng or true *)
	assertionIsWrong		:BOOL;
	(* contains the format string for the test message *)
	message					:Tc2_System.T_MaxString;
	(* TwinCAT printf with the test message *)
	messageStringBuilder	:Tc2_Utilities.FB_FormatString;
	(* return value of Tc2_System.F_CheckMemoryArea *)
	memoryArea				:Tc2_System.E_TcMemoryArea;
	(*  return value of Tc2_System.F_CheckMemoryArea as string *)
	areaString				:Tc2_System.T_MaxString;
END_VAR
THIS^.assertorContainer.resetAssertor();

memoryArea	:= Tc2_System.F_CheckMemoryArea(address, sizeInBytes);
areaString	:= THIS^.memoryAreaToString(memoryArea);
assertionIsWrong := (memoryArea <> Tc2_System.E_TcMemoryArea.Unknown);

message := SEL(
	assertionIsWrong,
	'address is 16#%X ($'%s$') sizeInBytes is %d return value of Tc2_System.F_CheckMemoryArea is $'%s$' assertion must be TRUE', 
	'address is 16#%X ($'%s$') sizeInBytes is %d return value of Tc2_System.F_CheckMemoryArea is $'%s$' assertion must be FALSE'
);
messageStringBuilder(
	sFormat := message,
	arg1 := THIS^.AnyToArg(address),
	arg2 := THIS^.AnyToArg(symbol),
	arg3 := THIS^.AnyToArg(sizeInBytes),
	arg4 := THIS^.AnyToArg(areaString)
);

THIS^.assertorContainer.assertor.assert.pointers.memoryAreaIsUnkown(
	address := address,
	sizeInBytes := sizeInBytes,
	message := ''
);

THIS^.AssertEquals_BOOL(
	Expected 	:= assertionIsWrong,
	Actual 		:= THIS^.assertorContainer.wasAssertionWrong,
	Message 	:= messageStringBuilder.sOut
);
END_METHOD

(*

short summary
==================
This test method tests ``assert.pointers.isNotEqualTo``
method of CNM_AssertionInterfaceLib library, 
it provides the possibility to handover test data via parameter 


.. <legal notes>

legal notes
=================
| SPDX-FileCopyrightText: © 2022 ekvip automation GmbH <info@ekvip.de>
| SPDX-License-Identifier: Apache-2.0
| For details check: Apache-2.0_

.. _Apache-2.0: https://www.apache.org/licenses/LICENSE-2.0

.. </legal notes>

parameters
==========

*)

METHOD testNotIsEqualTo
VAR_INPUT
	(* for the test it's the parameter ``address1`` *)
	address1	:PVOID;
	(* for the test it's the parameter ``address2`` *)
	address2	:PVOID;
END_VAR
VAR
	(* just the expectation if the assertion to test must be worng or true *)
	assertionIsWrong		:BOOL;
	(* contains the format string for the test message *)
	message					:Tc2_System.T_MaxString;
	(* TwinCAT printf with the test message *)
	messageStringBuilder	:Tc2_Utilities.FB_FormatString;
END_VAR
THIS^.assertorContainer.resetAssertor();

assertionIsWrong := (address1 = address2);
message := SEL(
	assertionIsWrong,
	'address1 is 16#%X address2 is 16#%X assertion must be TRUE', 
	'address1 is 16#%X address2 is 16#%X assertion must be FALSE'
);
messageStringBuilder(
	sFormat := message,
	arg1 := THIS^.AnyToArg(address1),
	arg2 := THIS^.AnyToArg(address2)
);

THIS^.assertorContainer.assertor.assert.pointers.isNotEqualTo(
	address1 := address1,
	address2 := address2,
	message := ''
);

THIS^.AssertEquals_BOOL(
	Expected 	:= assertionIsWrong,
	Actual 		:= THIS^.assertorContainer.wasAssertionWrong,
	Message 	:= messageStringBuilder.sOut
);
END_METHOD

END_FUNCTION_BLOCK

// ---- AssertionTester/AssertionTests/StringAssertions/StringAssertionTests.TcPOU
(*

short summary
=============

.. <legal notes>

legal notes
=================
| SPDX-FileCopyrightText: © 2023 ekvip automation GmbH <info@ekvip.de>
| SPDX-License-Identifier: Apache-2.0
| For details check: Apache-2.0_

.. _Apache-2.0: https://www.apache.org/licenses/LICENSE-2.0

.. </legal notes>

methods and properties
======================

*)

{warning 'header is generated please add your documentation'}
FUNCTION_BLOCK StringAssertionTests EXTENDS AbstractAssertorTest

VAR
	testDataStringLengthIsExact 	: ARRAY[0 ..IsLengthTestDataSet.SIZE_OF_IS_DATASET] OF IsLengthBasicData;
	testDataStringContains 			: ARRAY[0..containsTestDataSet.SIZE_OF_CONTAINS_DATASET] OF containsDataStr;
	testDataStringContainsNo 		: ARRAY[0..containsNOTestDataSet.SIZE_OF_CONTAINSNO_DATASET] OF containsDataStr;
	testDataStringStartsWith		: ARRAY[0..startsWithDataSet.SIZE_OF_STARTWITH_DATASET] OF containsDataStr;
	testDataStringEndsWith 			: ARRAY[0..endsWithDataSet.SIZE_OF_ENDSWITH_DATASET] OF containsDataStr;
	testDataStringIsEqual			: ARRAY[0..isEqualToTestDataSet.SIZE_OF_ISEQUALTO_DATASET] OF isEqualToDataStr;
	testDataStringIsNotEqual		: ARRAY[0..isNotEqualToTestDataSet.SIZE_OF_ISNOTEQUALTO_DATASET] OF isEqualToDataStr;
	testDataStringIsEmpty			: ARRAY[0..isEmptyTestDataSet.SIZE_OF_ISEMPTY_DATASET] OF isEmptyDataStr;
	testDataStringIsNotEmpty		: ARRAY[0..isNotEmtyTestDataSet.SIZE_OF_ISNOTEMPTY_DATASET] OF isEmptyDataStr;
	testDataStringIsLenghtBetween	: ARRAY[0..IsLengthBetweenDataSet.SIZE_OF_LENGTHBETWEEN_DATASET] OF IsLengthBetweenBasicData;
	
END_VAR

testAnyString_isEmpty();
testAnyString_isNotEmpty();
testAnyString_isEqualTo();
testAnyString_isNotEqualTo();
testAnyString_lengthIsExact();


THIS^.runTestIsLength();
THIS^.runTestContains();
THIS^.runTestContainsNo();
THIS^.runTestEndsWith();
THIS^.runTestStartsWith();
THIS^.runTestIsEmpty();
THIS^.runTestIsNotEmpty();
THIS^.runTestIsEqualTo();
THIS^.runTestIsNotEqualTo();
THIS^.runTestLengthIsBetween();

(*

short summary
=============

.. <legal notes>

legal notes
=================
| SPDX-FileCopyrightText: © 2023 ekvip automation GmbH <info@ekvip.de>
| SPDX-License-Identifier: Apache-2.0
| For details check: Apache-2.0_

.. _Apache-2.0: https://www.apache.org/licenses/LICENSE-2.0

.. </legal notes>

parameters
==========

*)

{warning 'header is generated please add your documentation'}
METHOD FB_init : BOOL
VAR_INPUT
    bInitRetains : BOOL; // if TRUE, the retain variables are initialized (warm start / cold start)
    bInCopyCode : BOOL;  // if TRUE, the instance afterwards gets moved into the copy code (online change)
	classToBeTested :IAssertorContainer;
END_VAR
THIS^.testDataStringLengthIsExact 	:= IsLengthTestDataSet.IsLenghtDataSetCommon;
THIS^.testDataStringContains 		:= containsTestDataSet.containsDataSetCommon;	
THIS^.testDataStringContainsNo		:= containsNoTestDataSet.containsNoDataSetCommon;
THIS^.testDataStringEndsWith		:= endsWithDataSet.endsWithDataSetCommon;
THIS^.testDataStringStartsWith		:= startsWithDataSet.StartsWithDataSetCommon;
THIS^.testDataStringIsEqual			:= isEqualToTestDataSet.isEqualToDataSetCommon;		
THIS^.testDataStringIsNotEqual		:= isNotEqualToTestDataSet.isNotEqualDataSetCommon;
THIS^.testDataStringIsEmpty			:= isEmptyTestDataSet.isEmptyDataSetCommon;
THIS^.testDataStringIsNotEmpty		:= isNotEmtyTestDataSet.isNotEmptyDataSetCommon;
THIS^.testDataStringIsLenghtBetween	:= IsLengthBetweenDataSet.isLenghtBetweenToDataSetCommon;
END_METHOD

(*

short summary
=============

.. <legal notes>

legal notes
=================
| SPDX-FileCopyrightText: © 2023 ekvip automation GmbH <info@ekvip.de>
| SPDX-License-Identifier: Apache-2.0
| For details check: Apache-2.0_

.. _Apache-2.0: https://www.apache.org/licenses/LICENSE-2.0

.. </legal notes>

parameters
==========

*)

{warning 'header is generated please add your documentation'}
METHOD reset
VAR_INPUT
END_VAR
THIS^.assertorContainer.resetAssertor();
END_METHOD

(*

short summary
=============

.. <legal notes>

legal notes
=================
| SPDX-FileCopyrightText: © 2023 ekvip automation GmbH <info@ekvip.de>
| SPDX-License-Identifier: Apache-2.0
| For details check: Apache-2.0_

.. _Apache-2.0: https://www.apache.org/licenses/LICENSE-2.0

.. </legal notes>

parameters
==========

*)

{warning 'header is generated please add your documentation'}
METHOD runTestContains
VAR
	testDataIterator	:USINT;
END_VAR
TEST('ContainsTests');
FOR testDataIterator := 0 TO containsTestDataSet.SIZE_OF_contains_DATASET DO
	IF (THIS^.testDataStringContains[testDataIterator].typeToTest = TypeToTest.TEST_STRING) THEN
		
		THIS^.testAnyStringContains(THIS^.testDataStringContains[testDataIterator], testDataIterator);
		THIS^.testAsciiStringContains (THIS^.testDataStringContains[testDataIterator], testDataIterator);
		
	ELSIF (THIS^.testDataStringContains[testDataIterator].typeToTest = TypeToTest.TEST_WSTRING) THEN
		
		THIS^.testAnyStringContains(THIS^.testDataStringContains[testDataIterator], testDataIterator);
		THIS^.testUtf16StringContains(THIS^.testDataStringContains[testDataIterator], testDataIterator);
		
	END_IF;
END_FOR

TEST_FINISHED();
END_METHOD

(*

short summary
=============

.. <legal notes>

legal notes
=================
| SPDX-FileCopyrightText: © 2023 ekvip automation GmbH <info@ekvip.de>
| SPDX-License-Identifier: Apache-2.0
| For details check: Apache-2.0_

.. _Apache-2.0: https://www.apache.org/licenses/LICENSE-2.0

.. </legal notes>

parameters
==========

*)

{warning 'header is generated please add your documentation'}
METHOD runTestContainsNo
VAR
	testDataIterator	:USINT;
END_VAR
TEST('ContainsNoTests');
FOR testDataIterator:= 0 TO containsNoTestDataSet.SIZE_OF_containsNo_DATASET DO
	IF (THIS^.testDataStringContainsNo[testDataIterator].typeToTest = TypeToTest.TEST_STRING) THEN
		
		THIS^.testAnyStringContainsNo(THIS^.testDataStringContainsno[testDataIterator], testDataIterator);
		THIS^.testAsciiStringContainsNo (THIS^.testDataStringContainsno[testDataIterator], testDataIterator);
		
	ELSIF (THIS^.testDataStringContainsNo[testDataIterator].typeToTest = TypeToTest.TEST_WSTRING) THEN
		
		THIS^.testAnyStringContainsNo(THIS^.testDataStringContainsno[testDataIterator], testDataIterator);
		THIS^.testUtf16StringContainsNo(THIS^.testDataStringContainsno[testDataIterator], testDataIterator);
		
	END_IF;
END_FOR

TEST_FINISHED();
END_METHOD

(*

short summary
=============

.. <legal notes>

legal notes
=================
| SPDX-FileCopyrightText: © 2023 ekvip automation GmbH <info@ekvip.de>
| SPDX-License-Identifier: Apache-2.0
| For details check: Apache-2.0_

.. _Apache-2.0: https://www.apache.org/licenses/LICENSE-2.0

.. </legal notes>

parameters
==========

*)

{warning 'header is generated please add your documentation'}
METHOD runTestEndsWith
VAR
	testDataIterator	: USINT;
END_VAR
TEST('endsWithTests');

FOR testDataIterator := 0 TO endsWithDataSet.SIZE_OF_ENDSWITH_DATASET DO
	IF (THIS^.testDataStringEndsWith[testDataIterator].typeToTest = TypeToTest.TEST_STRING) THEN
		
		THIS^.testAnyStringEndsWith(THIS^.testDataStringEndsWith[testDataIterator], testDataIterator);
		THIS^.testAsciiEndsWith(THIS^.testDataStringEndsWith[testDataIterator], testDataIterator);
		
	ELSIF (THIS^.testDataStringEndsWith[testDataIterator].typeToTest = TypeToTest.TEST_WSTRING) THEN
		
		THIS^.testAnyStringEndsWith(THIS^.testDataStringEndsWith[testDataIterator], testDataIterator);
		THIS^.testUtf16EndsWith(THIS^.testDataStringEndsWith[testDataIterator], testDataIterator);
		
	END_IF;
END_FOR

TEST_FINISHED();
END_METHOD

(*

short summary
=============

.. <legal notes>

legal notes
=================
| SPDX-FileCopyrightText: © 2023 ekvip automation GmbH <info@ekvip.de>
| SPDX-License-Identifier: Apache-2.0
| For details check: Apache-2.0_

.. _Apache-2.0: https://www.apache.org/licenses/LICENSE-2.0

.. </legal notes>

parameters
==========

*)

{warning 'header is generated please add your documentation'}
METHOD runTestIsEmpty
VAR
	testDataIterator	: USINT;
END_VAR
TEST('isEmptyTests');

FOR testDataIterator := 0 TO isEmptyTestDataSet.SIZE_OF_ISEMPTY_DATASET DO
	IF (THIS^.testDataStringIsEmpty[testDataIterator].typeToTest = TypeToTest.TEST_STRING) THEN
		
		THIS^.testAnyStringIsEmpty(THIS^.testDataStringIsEmpty[testDataIterator], testDataIterator);
		THIS^.testAsciiIsEmpty(THIS^.testDataStringIsEmpty[testDataIterator], testDataIterator);
		
	ELSIF (THIS^.testDataStringIsEmpty[testDataIterator].typeToTest = TypeToTest.TEST_WSTRING) THEN
		
		THIS^.testAnyStringIsEmpty(THIS^.testDataStringIsEmpty[testDataIterator], testDataIterator);
		THIS^.testUtf16IsEmpty(THIS^.testDataStringIsEmpty[testDataIterator], testDataIterator);
		
	END_IF;
END_FOR

TEST_FINISHED();
END_METHOD

(*

short summary
=============

.. <legal notes>

legal notes
=================
| SPDX-FileCopyrightText: © 2023 ekvip automation GmbH <info@ekvip.de>
| SPDX-License-Identifier: Apache-2.0
| For details check: Apache-2.0_

.. _Apache-2.0: https://www.apache.org/licenses/LICENSE-2.0

.. </legal notes>

parameters
==========

*)

{warning 'header is generated please add your documentation'}
METHOD runTestIsEqualTo
VAR
	testDataIterator	: USINT;
END_VAR
TEST('isEqualToTests');

FOR testDataIterator := 0 TO isEqualToTestDataSet.SIZE_OF_ISEQUALTO_DATASET DO
	IF (THIS^.testDataStringIsEqual[testDataIterator].typeToTest = TypeToTest.TEST_STRING) THEN
		
		THIS^.testAnyStringIsEqualTo(THIS^.testDataStringIsEqual[testDataIterator], testDataIterator);
		THIS^.testAsciiIsEqualTo(THIS^.testDataStringIsEqual[testDataIterator], testDataIterator);
		
	ELSIF (THIS^.testDataStringIsEqual[testDataIterator].typeToTest = TypeToTest.TEST_WSTRING) THEN
		
		THIS^.testAnyStringIsEqualTo(THIS^.testDataStringIsEqual[testDataIterator], testDataIterator);
		THIS^.testUtf16IsEqualTo(THIS^.testDataStringIsEqual[testDataIterator], testDataIterator);
		
	END_IF;
END_FOR

TEST_FINISHED();
END_METHOD

(*

short summary
=============

.. <legal notes>

legal notes
=================
| SPDX-FileCopyrightText: © 2023 ekvip automation GmbH <info@ekvip.de>
| SPDX-License-Identifier: Apache-2.0
| For details check: Apache-2.0_

.. _Apache-2.0: https://www.apache.org/licenses/LICENSE-2.0

.. </legal notes>

parameters
==========

*)

{warning 'header is generated please add your documentation'}
METHOD runTestIsLength
VAR
	testDataIterator	:USINT;
END_VAR
TEST('IsLenghtIsTests');
FOR testDataIterator:= 0 TO IsLengthTestDataSet.SIZE_OF_IS_DATASET DO
	IF (THIS^.testDataStringLengthIsExact[testDataIterator].typeToTest = TypeToTest.TEST_STRING) THEN
		
		THIS^.testAnyStringLengthIs(THIS^.testDataStringLengthIsExact[testDataIterator], testDataIterator);
		THIS^.testAsciiStringlengthIs (THIS^.testDataStringLengthIsExact[testDataIterator], testDataIterator);
		
	ELSIF (THIS^.testDataStringLengthIsExact[testDataIterator].typeToTest = TypeToTest.TEST_WSTRING) THEN
		
		THIS^.testAnyStringLengthIs(THIS^.testDataStringLengthIsExact[testDataIterator], testDataIterator);
		THIS^.testUtf16StringlengthIs(THIS^.testDataStringLengthIsExact[testDataIterator], testDataIterator);
		
	END_IF;
END_FOR

TEST_FINISHED();
END_METHOD

(*

short summary
=============

.. <legal notes>

legal notes
=================
| SPDX-FileCopyrightText: © 2023 ekvip automation GmbH <info@ekvip.de>
| SPDX-License-Identifier: Apache-2.0
| For details check: Apache-2.0_

.. _Apache-2.0: https://www.apache.org/licenses/LICENSE-2.0

.. </legal notes>

parameters
==========

*)

{warning 'header is generated please add your documentation'}
METHOD runTestIsNotEmpty
VAR
	testDataIterator	: USINT;
END_VAR
TEST('isNotEmptyTests');

FOR testDataIterator := 0 TO isNotEmtyTestDataSet.SIZE_OF_ISNOTEMPTY_DATASET DO
	IF (THIS^.testDataStringIsNotEmpty[testDataIterator].typeToTest = TypeToTest.TEST_STRING) THEN
		
		THIS^.testAnyStringIsNotEmpty(THIS^.testDataStringIsNotEmpty[testDataIterator], testDataIterator);
		THIS^.testAsciiIsNotEmpty(THIS^.testDataStringIsNotEmpty[testDataIterator], testDataIterator);
		
	ELSIF (THIS^.testDataStringIsNotEmpty[testDataIterator].typeToTest = TypeToTest.TEST_WSTRING) THEN
		
		THIS^.testAnyStringIsNotEmpty(THIS^.testDataStringIsNotEmpty[testDataIterator], testDataIterator);
		THIS^.testUtf16IsNotEmpty(THIS^.testDataStringIsNotEmpty[testDataIterator], testDataIterator);
		
	END_IF;
END_FOR

TEST_FINISHED();
END_METHOD

(*

short summary
=============

.. <legal notes>

legal notes
=================
| SPDX-FileCopyrightText: © 2023 ekvip automation GmbH <info@ekvip.de>
| SPDX-License-Identifier: Apache-2.0
| For details check: Apache-2.0_

.. _Apache-2.0: https://www.apache.org/licenses/LICENSE-2.0

.. </legal notes>

parameters
==========

*)

{warning 'header is generated please add your documentation'}
METHOD runTestIsNotEqualTo
VAR
	testDataIterator	: USINT;
END_VAR
TEST('isNotEqualToTests');

FOR testDataIterator := 0 TO isNotEqualToTestDataSet.SIZE_OF_ISNOTEQUALTO_DATASET DO
	IF (THIS^.testDataStringIsNotEqual[testDataIterator].typeToTest = TypeToTest.TEST_STRING) THEN
		
		THIS^.testAnyStringIsNotEqualTo(THIS^.testDataStringIsNotEqual[testDataIterator], testDataIterator);
		THIS^.testAsciiIsNotEqualTo(THIS^.testDataStringIsNotEqual[testDataIterator], testDataIterator);
		
	ELSIF (THIS^.testDataStringIsNotEqual[testDataIterator].typeToTest = TypeToTest.TEST_WSTRING) THEN
		
		THIS^.testAnyStringIsNotEqualTo(THIS^.testDataStringIsNotEqual[testDataIterator], testDataIterator);
		THIS^.testUtf16IsNotEqualTo(THIS^.testDataStringIsNotEqual[testDataIterator], testDataIterator);
		
	END_IF;
END_FOR

TEST_FINISHED();
END_METHOD

(*

short summary
=============

.. <legal notes>

legal notes
=================
| SPDX-FileCopyrightText: © 2023 ekvip automation GmbH <info@ekvip.de>
| SPDX-License-Identifier: Apache-2.0
| For details check: Apache-2.0_

.. _Apache-2.0: https://www.apache.org/licenses/LICENSE-2.0

.. </legal notes>

parameters
==========

*)

{warning 'header is generated please add your documentation'}
METHOD runTestLengthIsBetween : BOOL
VAR
	testDataIterator	:USINT;
END_VAR
TEST('IsLenghtBetweenTests');
FOR testDataIterator:= 0 TO IsLengthBetweenDataSet.SIZE_OF_LENGTHBETWEEN_DATASET DO
	IF (THIS^.testDataStringIsLenghtBetween[testDataIterator].typeToTest = TypeToTest.TEST_STRING) THEN
		
		THIS^.testAnyStringLengthBetween(THIS^.testDataStringIsLenghtBetween[testDataIterator], testDataIterator);
		THIS^.testAsciiStringLengthBetween (THIS^.testDataStringIsLenghtBetween[testDataIterator], testDataIterator);
		
	ELSIF (THIS^.testDataStringIsLenghtBetween[testDataIterator].typeToTest = TypeToTest.TEST_WSTRING) THEN
		
		THIS^.testAnyStringLengthBetween(THIS^.testDataStringIsLenghtBetween[testDataIterator], testDataIterator);
		THIS^.testUtf16StringLengthBetween(THIS^.testDataStringIsLenghtBetween[testDataIterator], testDataIterator);
		
	END_IF;
END_FOR

TEST_FINISHED();
END_METHOD

(*

short summary
=============

.. <legal notes>

legal notes
=================
| SPDX-FileCopyrightText: © 2023 ekvip automation GmbH <info@ekvip.de>
| SPDX-License-Identifier: Apache-2.0
| For details check: Apache-2.0_

.. _Apache-2.0: https://www.apache.org/licenses/LICENSE-2.0

.. </legal notes>

parameters
==========

*)

{warning 'header is generated please add your documentation'}
METHOD runTestStartsWith
VAR
	testDataIterator	: USINT;
END_VAR
TEST('StartsWithTests');
FOR testDataIterator := 0 TO startsWithDataSet.SIZE_OF_STARTWITH_DATASET DO
	IF (THIS^.testDataStringStartsWith[testDataIterator].typeToTest = TypeToTest.TEST_STRING) THEN
		
		THIS^.testAnyStringStartsWith(THIS^.testDataStringStartsWith[testDataIterator], testDataIterator);
		THIS^.testAsciiStartsWith(THIS^.testDataStringStartsWith[testDataIterator], testDataIterator);
		
	ELSIF (THIS^.testDataStringStartsWith[testDataIterator].typeToTest = TypeToTest.TEST_WSTRING) THEN
		
		THIS^.testAnyStringStartsWith(THIS^.testDataStringStartsWith[testDataIterator], testDataIterator);
		THIS^.testUtf16StartsWith(THIS^.testDataStringStartsWith[testDataIterator], testDataIterator);
		
	END_IF;
END_FOR

TEST_FINISHED();
END_METHOD

(*

short summary
=============

.. <legal notes>

legal notes
=================
| SPDX-FileCopyrightText: © 2023 ekvip automation GmbH <info@ekvip.de>
| SPDX-License-Identifier: Apache-2.0
| For details check: Apache-2.0_

.. _Apache-2.0: https://www.apache.org/licenses/LICENSE-2.0

.. </legal notes>

parameters
==========

*)

{warning 'header is generated please add your documentation'}
METHOD testAnyString_isEmpty

VAR 
  testString1: STRING(50);
  testString2: STRING;
  number: INT;
END_VAR

// anyStringAssertionTests.isEmpty Tests

//-------------------------------------------------------------------------------------------------------
TEST('anyStringAssertionTest.isEmpty with stringToCheck:= emptyString');

testString1:= '';
THIS^.assertorContainer.resetAssertor();
THIS^.assertorContainer.assertor.assert.strings.anyString.isEmpty(
  stringToCheck := testString1,
  message := ''
);
THIS^.AssertFalse(
	Condition := THIS^.assertorContainer.wasAssertionWrong,
	Message := 'anyStringAssertionTests.isEmpty assertion shall be wrong, stringToCheck:= emptyString '
);
TEST_FINISHED();

//-------------------------------------------------------------------------------------------------------

TEST('anyStringAssertionTest.isEmpty with stringToCheck:= space');

testString1:= ' ';
THIS^.assertorContainer.resetAssertor();
THIS^.assertorContainer.assertor.assert.strings.anyString.isEmpty(
  stringToCheck := testString1,
  message := ''
);
THIS^.AssertTrue(
	Condition := THIS^.assertorContainer.wasAssertionWrong,
	Message := 'anyStringAssertionTests.isEmpty assertion shall be wrong, stringToCheck:= just space'
);
TEST_FINISHED();

//-------------------------------------------------------------------------------------------------------

TEST('anyStringAssertionTest.isEmpty with stringToCheck:= point');

testString1:= '.';
THIS^.assertorContainer.resetAssertor();
THIS^.assertorContainer.assertor.assert.strings.anyString.isEmpty(
  stringToCheck := testString1,
  message := ''
);
THIS^.AssertTrue(
	Condition := THIS^.assertorContainer.wasAssertionWrong,
	Message := 'anyStringAssertionTests.isEmpty assertion shall be wrong, stringToCheck:= point'
);
TEST_FINISHED();

//-------------------------------------------------------------------------------------------------------

TEST('anyStringAssertionTest.isEmpty with stringToCheck:= emptyStringVar');

testString1:= testString2;
THIS^.assertorContainer.resetAssertor();
THIS^.assertorContainer.assertor.assert.strings.anyString.isEmpty(
  stringToCheck := testString1,
  message := ''
);
THIS^.AssertFalse(
	Condition := THIS^.assertorContainer.wasAssertionWrong,
	Message := 'anyStringAssertionTests.isEmpty assertion shall be wrong, stringToCheck:= emptyStringVar'
);
TEST_FINISHED();

//-------------------------------------------------------------------------------------------------------

TEST('anyStringAssertionTest.isEmpty with stringToCheck:= wierdString');

testString1:= 'sadhasdhasduhuiashdui';
THIS^.assertorContainer.resetAssertor();
THIS^.assertorContainer.assertor.assert.strings.anyString.isEmpty(
  stringToCheck := testString1,
  message := ''
);
THIS^.AssertTrue(
	Condition := THIS^.assertorContainer.wasAssertionWrong,
	Message := 'anyStringAssertionTests.isEmpty assertion shall be wrong, stringToCheck:= emptyStringVar'
);
TEST_FINISHED();

//-------------------------------------------------------------------------------------------------------

TEST('anyStringAssertionTest.isEmpty with stringToCheck:=   +gdjsnd.8959889mfknfji');

testString1:= '   +gdjsnd.8959889mfknfji';
THIS^.assertorContainer.resetAssertor();
THIS^.assertorContainer.assertor.assert.strings.anyString.isEmpty(
  stringToCheck := testString1,
  message := ''
);
THIS^.AssertTrue(
	Condition := THIS^.assertorContainer.wasAssertionWrong,
	Message := 'anyStringAssertionTests.isEmpty assertion shall be wrong, stringToCheck:= emptyStringVar'
);
TEST_FINISHED();

//-------------------------------------------------------------------------------------------------------

TEST('anyStringAssertionTest.isEmpty with stringToCheck:=   converted int');

testString1:= INT_TO_STRING(number);
THIS^.assertorContainer.resetAssertor();
THIS^.assertorContainer.assertor.assert.strings.anyString.isEmpty(
  stringToCheck := testString1,
  message := ''
);
THIS^.AssertTrue(
	Condition := THIS^.assertorContainer.wasAssertionWrong,
	Message := 'anyStringAssertionTests.isEmpty assertion shall be wrong, stringToCheck:=  converted int'
);
TEST_FINISHED();
END_METHOD

(*

short summary
=============

.. <legal notes>

legal notes
=================
| SPDX-FileCopyrightText: © 2023 ekvip automation GmbH <info@ekvip.de>
| SPDX-License-Identifier: Apache-2.0
| For details check: Apache-2.0_

.. _Apache-2.0: https://www.apache.org/licenses/LICENSE-2.0

.. </legal notes>

parameters
==========

*)

{warning 'header is generated please add your documentation'}
METHOD testAnyString_isEqualTo

VAR 
  testString1: STRING(50);
  testString2: STRING(30);
  testString3: WSTRING(50);
  testString4: STRING(50);
  testString5: WSTRING(400);
  testString6: WSTRING(400);
  number: INT;
END_VAR

// anyStringAssertionTests.isEqualTo Tests

//-------------------------------------------------------------------------------------------------------
TEST('anyStringAssertionTest.isEqualTo with stringToCheck:= emptyString , expected:= emptyString , ignoreCases:= TRUE ,');

THIS^.assertorContainer.resetAssertor();
THIS^.assertorContainer.assertor.assert.strings.anyString.isEqualTo(
  stringToCheck:= testString1 , 
  expected:= testString2 ,
  ignoreCases:= TRUE ,
  message:='' );
  
THIS^.AssertFalse(
	Condition := THIS^.assertorContainer.wasAssertionWrong,
	Message := 'anyStringAssertionTests.isEqualTo , stringToCheck:= emptyString , expected:= emptyString , ignoreCases:= TRUE '
);
TEST_FINISHED();

//-------------------------------------------------------------------------------------------------------
TEST('anyStringAssertionTest.isEqualTo with stringToCheck:= emptyString assign , expected:= emptyString assign , ignoreCases:= TRUE ,');

testString1:= '';
testString2:= '';

THIS^.assertorContainer.resetAssertor();
THIS^.assertorContainer.assertor.assert.strings.anyString.isEqualTo(
  stringToCheck:= testString1 , 
  expected:= testString2 ,
  ignoreCases:= TRUE ,
  message:='' );
  
THIS^.AssertFalse(
	Condition := THIS^.assertorContainer.wasAssertionWrong,
	Message := 'anyStringAssertionTests.isEqualTo , stringToCheck:= emptyString assign, expected:= emptyString assign , ignoreCases:= TRUE '
);
TEST_FINISHED();

//-------------------------------------------------------------------------------------------------------
TEST('anyStringAssertionTest.isEqualTo with stringToCheck:= abcd56ä² , expected:= abcd56ä2 , ignoreCases:= TRUE ,');

testString1:= 'abcd56ä²';
testString2:= 'abcd56ä2';

THIS^.assertorContainer.resetAssertor();
THIS^.assertorContainer.assertor.assert.strings.anyString.isEqualTo(
  stringToCheck:= testString1 , 
  expected:= testString2 ,
  ignoreCases:= TRUE ,
  message:='' );
  
THIS^.AssertTrue(
	Condition := THIS^.assertorContainer.wasAssertionWrong,
	Message := 'anyStringAssertionTests.isEqualTo assertion shall be wrong, stringToCheck:= abcd56ä²  , expected:= abcd56ä2 , ignoreCases:= TRUE'
);
TEST_FINISHED();


//-------------------------------------------------------------------------------------------------------
TEST('anyStringAssertionTest.isEqualTo with stringToCheck:= abcd56ä²  , expected:= abcd56ä2 , ignoreCases:= False ,');

testString1:= 'abcd56ä²';
testString2:= 'abcd56ä2';

THIS^.assertorContainer.resetAssertor();
THIS^.assertorContainer.assertor.assert.strings.anyString.isEqualTo(
  stringToCheck:= testString1 , 
  expected:= testString2 ,
  ignoreCases:= FALSE ,
  message:='' );
  
THIS^.AssertTrue(
	Condition := THIS^.assertorContainer.wasAssertionWrong,
	Message := 'anyStringAssertionTests.isEqualTo assertion shall be wrong, stringToCheck:= abcd56ä²  , expected:= abcd56ä2 , ignoreCases:= false'
);
TEST_FINISHED();

//-------------------------------------------------------------------------------------------------------
TEST('anyStringAssertionTest.isEqualTo with stringToCheck:= abc d56ä2  , expected:= abc  d56ä2 , ignoreCases:= TRUE ,');

testString1:= 'abc d56ä2';
testString2:= 'abc  d56ä2';

THIS^.assertorContainer.resetAssertor();
THIS^.assertorContainer.assertor.assert.strings.anyString.isEqualTo(
  stringToCheck:= testString1 , 
  expected:= testString2 ,
  ignoreCases:= TRUE ,
  message:='' );
  
THIS^.AssertTrue(
	Condition := THIS^.assertorContainer.wasAssertionWrong,
	Message := 'anyStringAssertionTests.isEqualTo , stringToCheck:= abc d56ä2  , expected:= abc  d56ä2 , ignoreCases:= TRUE ,'
);
TEST_FINISHED();

//-------------------------------------------------------------------------------------------------------
TEST('anyStringAssertionTest.isEqualTo with stringToCheck:= abcd56ä2&§ (string) , expected:= abcd56ä2&§ (wstring), ignoreCases:= TRUE ,');

testString1:= 'abcd56ä2&§';
testString3:= "abcd56ä2&§";

THIS^.assertorContainer.resetAssertor();
THIS^.assertorContainer.assertor.assert.strings.anyString.isEqualTo(
  stringToCheck:= testString1 , 
  expected:= testString3 ,
  ignoreCases:= TRUE ,
  message:='' );
  
THIS^.AssertTrue(
	Condition := THIS^.assertorContainer.wasAssertionWrong,
	Message := 'anyStringAssertionTests.isEqualTo stringToCheck:= abcd56ä2&§ (string) , expected:= abcd56ä2&§ (wstring) , ignoreCases:= TRUE'
);
TEST_FINISHED();

//-------------------------------------------------------------------------------------------------------
TEST('anyStringAssertionTest.isEqualTo with stringToCheck:= abcd56ä2&§ (string) , expected:= abcd56ä2&§ (converted string)   , ignoreCases:= TRUE ,');

testString1:= 'abcd56ä2&§';
testString3:= "abcd56ä2&§";
testString4:= WSTRING_TO_STRING(testString3);

THIS^.assertorContainer.resetAssertor();
THIS^.assertorContainer.assertor.assert.strings.anyString.isEqualTo(
  stringToCheck:= testString1 , 
  expected:= testString4 ,
  ignoreCases:= TRUE ,
  message:='' );
  
THIS^.AssertFalse(
	Condition := THIS^.assertorContainer.wasAssertionWrong,
	Message := 'anyStringAssertionTests.isEqualTo stringToCheck:= abcd56ä2&§ (string) , expected:= expected:= abcd56ä2&§ (converted string) , ignoreCases:= TRUE'
);
TEST_FINISHED();


//-------------------------------------------------------------------------------------------------------
TEST('anyStringAssertionTest.isEqualTo with stringToCheck:= abcd56ä2&§ (string) , expected:= AbBd56ä2&§ , ignoreCases:= False ,');

testString1:= 'abcd56ä2&§';
testString2:='AbCd56ä2&§';

THIS^.assertorContainer.resetAssertor();
THIS^.assertorContainer.assertor.assert.strings.anyString.isEqualTo(
  stringToCheck:= testString1 , 
  expected:= testString2 ,
  ignoreCases:= TRUE ,
  message:='' );
  
THIS^.AssertFalse(
	Condition := THIS^.assertorContainer.wasAssertionWrong,
	Message := 'anyStringAssertionTests.isEqualTo with stringToCheck:= abcd56ä2&§  , expected:= AbBd56ä2&§ , ignoreCases:= False'
);
TEST_FINISHED();


//-------------------------------------------------------------------------------------------------------
TEST('anyStringAssertionTest.isEqualTo with stringToCheck:= äbcd56ä2&§ , expected:= äbcd56ä2&§ , ignoreCases:= False ,');

testString1:= 'abcd56ä2&§';
testString4:='äbcd56ä2&§';

THIS^.assertorContainer.resetAssertor();
THIS^.assertorContainer.assertor.assert.strings.anyString.isEqualTo(
  stringToCheck:= testString1 , 
  expected:= testString4 ,
  ignoreCases:= FALSE ,
  message:='' );
  
THIS^.AssertTrue(
	Condition := THIS^.assertorContainer.wasAssertionWrong,
	Message := 'anyStringAssertionTests.isEqualTo with stringToCheck:= abcd56ä2&§  , expected:= äbcd56ä2&§ , ignoreCases:= False'
);
TEST_FINISHED();

//-------------------------------------------------------------------------------------------------------
TEST('anyStringAssertionTest.isEqualTo with stringToCheck:= strange stuff arabic russian , expected:= strange stuff arabic russian , ignoreCases:= False ,');

testString5:= "иди сюда кусок дерьма ဒီကိုလာပါ ၊ تعال إلى هنا يا قطعة من الهراء";
testString6:="иди сюда кусок дерьма ဒီကိုလာပါ ၊ تعال إلى هنا يا قطعة من الهراء";

THIS^.assertorContainer.resetAssertor();
THIS^.assertorContainer.assertor.assert.strings.anyString.isEqualTo(
  stringToCheck:= testString5 , 
  expected:= testString6 ,
  ignoreCases:= FALSE ,
  message:='' );
  
THIS^.AssertFalse(
	Condition := THIS^.assertorContainer.wasAssertionWrong,
	Message := 'anyStringAssertionTests.isEqualTo with stringToCheck:= strange stuff arabic russian  , expected:= strange stuff arabic russian , ignoreCases:= False'
);
TEST_FINISHED();

//-------------------------------------------------------------------------------------------------------
TEST('anyStringAssertionTest.isEqualTo with stringToCheck:= strange stuff arabic russian 1 , expected:= strange stuff arabic russian 2, ignoreCases:= False ,');

testString5:= "иди сюд кусок дерьма ဒီကိုလာပါ ၊ تعال إلى هنا يا قطعة من الهراء";
testString6:="иди сюда кусок дерьма ဒီကိုလာပါ ၊ تعال إلى هنا يا قطعة من الهراء";

THIS^.assertorContainer.resetAssertor();
THIS^.assertorContainer.assertor.assert.strings.anyString.isEqualTo(
  stringToCheck:= testString5 , 
  expected:= testString6 ,
  ignoreCases:= FALSE ,
  message:='' );
  
THIS^.AssertTrue(
	Condition := THIS^.assertorContainer.wasAssertionWrong,
	Message := 'anyStringAssertionTests.isEqualTo with stringToCheck:= strange stuff arabic russian  , expected:= strange stuff arabic russian , ignoreCases:= False'
);
TEST_FINISHED();

//-------------------------------------------------------------------------------------------------------

TEST('anyStringAssertionTest.isEqualTo with stringToCheck:= strange stuff arabic russian capital , expected:= strange stuff arabic russian , ignoreCases:= true ,');

testString5:= "иди сюда Кусок дерьма ဒီကိုလာပါ ၊ تعال إلى هنا يا قطعة من الهراء";
testString6:="иди сюда кусок дерьма ဒီကိုလာပါ ၊ تعال إلى هنا يا قطعة من الهراء";

THIS^.assertorContainer.resetAssertor();
THIS^.assertorContainer.assertor.assert.strings.anyString.isEqualTo(
  stringToCheck:= testString5 , 
  expected:= testString6 ,
  ignoreCases:= TRUE ,
  message:='' );
  
THIS^.AssertFalse(
	Condition := THIS^.assertorContainer.wasAssertionWrong,
	Message := 'anyStringAssertionTests.isEqualTo with stringToCheck:= strange stuff arabic russian  , expected:= strange stuff arabic russian , ignoreCases:= true'
);
TEST_FINISHED();
END_METHOD

(*

short summary
=============

.. <legal notes>

legal notes
=================
| SPDX-FileCopyrightText: © 2023 ekvip automation GmbH <info@ekvip.de>
| SPDX-License-Identifier: Apache-2.0
| For details check: Apache-2.0_

.. _Apache-2.0: https://www.apache.org/licenses/LICENSE-2.0

.. </legal notes>

parameters
==========

*)

{warning 'header is generated please add your documentation'}
METHOD testAnyString_isNotEmpty

VAR
  testString1: STRING(50);
  testString2: STRING; 
END_VAR

// anyStringAssertionTests.isNotEmpty Tests

//-------------------------------------------------------------------------------------------------------
TEST('anyStringAssertionTest.isNotEmpty with stringToCheck:= emptyString');


testString1:= '';
THIS^.assertorContainer.resetAssertor();
THIS^.assertorContainer.assertor.assert.strings.anyString.isNOtEmpty(
  stringToCheck := testString1,
  message := ''
);
THIS^.AssertTrue(
	Condition := THIS^.assertorContainer.wasAssertionWrong,
	Message := 'anyStringAssertionTests.isNotEmpty assertion shall be wrong, stringToCheck:= emptyString '
);
TEST_FINISHED();

//-------------------------------------------------------------------------------------------------------

TEST('anyStringAssertionTest.isNotEmpty with stringToCheck:= space');

testString1:= ' ';
THIS^.assertorContainer.resetAssertor();
THIS^.assertorContainer.assertor.assert.strings.anyString.isNotEmpty(
  stringToCheck := testString1,
  message := ''
);
THIS^.AssertFalse(
	Condition := THIS^.assertorContainer.wasAssertionWrong,
	Message := 'anyStringAssertionTests.isNotEmpty assertion shall be wrong, stringToCheck:= just space'
);
TEST_FINISHED();

//-------------------------------------------------------------------------------------------------------

TEST('anyStringAssertionTest.isNotEmpty with stringToCheck:= point');

testString1:= '.';
THIS^.assertorContainer.resetAssertor();
THIS^.assertorContainer.assertor.assert.strings.anyString.isNotEmpty(
  stringToCheck := testString1,
  message := ''
);
THIS^.AssertFalse(
	Condition := THIS^.assertorContainer.wasAssertionWrong,
	Message := 'anyStringAssertionTests.isNotEmpty assertion shall be wrong, stringToCheck:= point'
);
TEST_FINISHED();

//-------------------------------------------------------------------------------------------------------

TEST('anyStringAssertionTest.isNotEmpty with stringToCheck:= emptyStringVar');

testString1:= testString2;
THIS^.assertorContainer.resetAssertor();
THIS^.assertorContainer.assertor.assert.strings.anyString.isNotEmpty(
  stringToCheck := testString1,
  message := ''
);
THIS^.AssertTrue(
	Condition := THIS^.assertorContainer.wasAssertionWrong,
	Message := 'anyStringAssertionTests.isNotEmpty assertion shall be wrong, stringToCheck:= emptyStringVar'
);
TEST_FINISHED();

//-------------------------------------------------------------------------------------------------------

TEST('anyStringAssertionTest.isNotEmpty with stringToCheck:= wierdString');

testString1:= 'sadhasdhasduhuiashdui';
THIS^.assertorContainer.resetAssertor();
THIS^.assertorContainer.assertor.assert.strings.anyString.isNotEmpty(
  stringToCheck := testString1,
  message := ''
);
THIS^.AssertFalse(
	Condition := THIS^.assertorContainer.wasAssertionWrong,
	Message := 'anyStringAssertionTests.isNotEmpty assertion shall be wrong, stringToCheck:= emptyStringVar'
);
TEST_FINISHED();

//-------------------------------------------------------------------------------------------------------

TEST('anyStringAssertionTest.isNotEmpty with stringToCheck:=   +gdjsnd.8959889mfknfji');

testString1:= '   +gdjsnd.8959889mfknfji';
THIS^.assertorContainer.resetAssertor();
THIS^.assertorContainer.assertor.assert.strings.anyString.isNotEmpty(
  stringToCheck := testString1,
  message := ''
);
THIS^.AssertFalse(
	Condition := THIS^.assertorContainer.wasAssertionWrong,
	Message := 'anyStringAssertionTests.isNotEmpty assertion shall be wrong, stringToCheck:= emptyStringVar'
);
TEST_FINISHED();
END_METHOD

(*

short summary
=============

.. <legal notes>

legal notes
=================
| SPDX-FileCopyrightText: © 2023 ekvip automation GmbH <info@ekvip.de>
| SPDX-License-Identifier: Apache-2.0
| For details check: Apache-2.0_

.. _Apache-2.0: https://www.apache.org/licenses/LICENSE-2.0

.. </legal notes>

parameters
==========

*)

{warning 'header is generated please add your documentation'}
METHOD testAnyString_isNotEqualTo 

VAR 
  testString1: STRING(50);
  testString2: STRING(30);
  testString3: WSTRING(50);
  testString4: STRING(50);
  testString5: WSTRING(400);
  testString6: WSTRING(400);
  number: INT;
END_VAR

// anyStringAssertionTests.isNotEqualTo Tests

//-------------------------------------------------------------------------------------------------------
TEST('anyStringAssertionTest.isNotEqualTo with stringToCheck:= emptyString , unexpected:= emptyString , ignoreCases:= TRUE ,');

THIS^.assertorContainer.resetAssertor();
THIS^.assertorContainer.assertor.assert.strings.anyString.isNotEqualTo(
  stringToCheck:= testString1 , 
  unexpected:= testString2 ,
  ignoreCases:= TRUE ,
  message:='' );
  
THIS^.AssertTrue(
	Condition := THIS^.assertorContainer.wasAssertionWrong,
	Message := 'anyStringAssertionTests.isNotEqualTo , stringToCheck:= emptyString , unexpected:= emptyString , ignoreCases:= TRUE'
);
TEST_FINISHED();


//-------------------------------------------------------------------------------------------------------
TEST('anyStringAssertionTest.isNotEqualTo with stringToCheck:= emptyString assign , unexpected:= emptyString assign , ignoreCases:= TRUE');

testString1:= '';
testString2:= '';

THIS^.assertorContainer.resetAssertor();
THIS^.assertorContainer.assertor.assert.strings.anyString.isNotEqualTo(
  stringToCheck:= testString1 , 
  unexpected:= testString2 ,
  ignoreCases:= TRUE ,
  message:='' );  
  
  
THIS^.AssertTrue(
	Condition := THIS^.assertorContainer.wasAssertionWrong,
	Message := 'anyStringAssertionTests.isNotEqualTo , stringToCheck:= emptyString assign, unexpected:= emptyString assign , ignoreCases:= TRUE');
TEST_FINISHED();

//-------------------------------------------------------------------------------------------------------

TEST('anyStringAssertionTest.isNotEqualTo with stringToCheck:= abcd56ä² , unexpected:= abcd56ä2 , ignoreCases:= TRUE ,');

testString1:= 'abcd56ä²';
testString2:= 'abcd56ä2';

THIS^.assertorContainer.resetAssertor();
THIS^.assertorContainer.assertor.assert.strings.anyString.isNotEqualTo(
  stringToCheck:= testString1 , 
  unexpected:= testString2 ,
  ignoreCases:= TRUE ,
  message:='' );
  
THIS^.AssertFalse(
	Condition := THIS^.assertorContainer.wasAssertionWrong,
	Message := 'anyStringAssertionTests.isNotEqualTo assertion shall be wrong, stringToCheck:= abcd56ä²  , unexpected:= abcd56ä2 , ignoreCases:= TRUE'
);
TEST_FINISHED();


//-------------------------------------------------------------------------------------------------------
TEST('anyStringAssertionTest.isEmpty with stringToCheck:= abcd56ä2  , unexpected:= abcd56ä2 , ignoreCases:= False ,');

testString1:= 'abcd56ä2';
testString2:= 'abcd56ä2';

THIS^.assertorContainer.resetAssertor();
THIS^.assertorContainer.assertor.assert.strings.anyString.isNotEqualTo(
  stringToCheck:= testString1 , 
  unexpected:= testString2 ,
  ignoreCases:= FALSE ,
  message:='' );
  
THIS^.AssertTrue(
	Condition := THIS^.assertorContainer.wasAssertionWrong,
	Message := 'anyStringAssertionTests.isNotEqualTo assertion shall be wrong, stringToCheck:= abcd56ä2  , unexpected:= abcd56ä2 , ignoreCases:= false'
);
TEST_FINISHED();


//-------------------------------------------------------------------------------------------------------
TEST('anyStringAssertionTest.isNotEqualTo with stringToCheck:= abc d56ä2  , unexpected:= abc  d56ä2 , ignoreCases:= TRUE ,');

testString1:= 'abc d56ä2';
testString2:= 'abc  d56ä2';

THIS^.assertorContainer.resetAssertor();
THIS^.assertorContainer.assertor.assert.strings.anyString.isnotEqualTo(
  stringToCheck:= testString1 , 
  unexpected:= testString2 ,
  ignoreCases:= TRUE ,
  message:='' );
  
THIS^.AssertFalse(
	Condition := THIS^.assertorContainer.wasAssertionWrong,
	Message := 'anyStringAssertionTests.isNotEqualTo , stringToCheck:= abc d56ä2  , unexpected:= abc  d56ä2 , ignoreCases:= TRUE ,'
);
TEST_FINISHED();

//-------------------------------------------------------------------------------------------------------
TEST('anyStringAssertionTest.isNotEqualTo with stringToCheck:= abcd56ä2&§ (string) , unexpected:= abcd56ä2&§ (wstring), ignoreCases:= TRUE ,');

testString1:= 'abcd56ä2&§';
testString3:= "abcd56ä2&§";

THIS^.assertorContainer.resetAssertor();
THIS^.assertorContainer.assertor.assert.strings.anyString.isNotEqualTo(
  stringToCheck:= testString1 , 
  unexpected:= testString3 ,
  ignoreCases:= TRUE ,
  message:='' );
  
THIS^.AssertFalse(
	Condition := THIS^.assertorContainer.wasAssertionWrong,
	Message := 'anyStringAssertionTests.isNotEqualTo stringToCheck:= abcd56ä2&§ (string) , unexpected:= abcd56ä2&§ (wstring) , ignoreCases:= TRUE'
);
TEST_FINISHED();

//-------------------------------------------------------------------------------------------------------
TEST('anyStringAssertionTest.isNotEqualTo with stringToCheck:= abcd56ä2&§ (string) , unexpected:= abcd56ä2&§ (converted string)   , ignoreCases:= TRUE ,');

testString1:= 'abcd56ä2&§';
testString3:= "abcd56ä2&§";
testString4:= WSTRING_TO_STRING(testString3);

THIS^.assertorContainer.resetAssertor();
THIS^.assertorContainer.assertor.assert.strings.anyString.isNotEqualTo(
  stringToCheck:= testString1 , 
  unexpected:= testString4 ,
  ignoreCases:= TRUE ,
  message:='' );
  
THIS^.AssertTrue(
	Condition := THIS^.assertorContainer.wasAssertionWrong,
	Message := 'anyStringAssertionTests.isNotEqualTo stringToCheck:= abcd56ä2&§ (string) , unexpected:= abcd56ä2&§ (converted string) , ignoreCases:= TRUE'
);
TEST_FINISHED();



//-------------------------------------------------------------------------------------------------------
TEST('anyStringAssertionTest.isNotEqualTo with stringToCheck:= abcd56ä2&§ (string) , unexpected:= AbBd56ä2&§ , ignoreCases:= False ,');

testString1:= 'abcd56ä2&§';
testString2:='AbCd56ä2&§';

THIS^.assertorContainer.resetAssertor();
THIS^.assertorContainer.assertor.assert.strings.anyString.isNotEqualTo(
  stringToCheck:= testString1 , 
  unexpected:= testString2 ,
  ignoreCases:= TRUE ,
  message:='' );
  
THIS^.AssertTrue(
	Condition := THIS^.assertorContainer.wasAssertionWrong,
	Message := 'anyStringAssertionTests.isNotEqualTo with stringToCheck:= abcd56ä2&§  , unexpected:= AbBd56ä2&§ , ignoreCases:= False'
);
TEST_FINISHED();


//-------------------------------------------------------------------------------------------------------
TEST('anyStringAssertionTest.isNotEqualTo with stringToCheck:= äbcd56ä2&§ , unexpected:= äbcd56ä2&§ , ignoreCases:= False ,');

testString1:= 'abcd56ä2&§';
testString4:='äbcd56ä2&§';

THIS^.assertorContainer.resetAssertor();
THIS^.assertorContainer.assertor.assert.strings.anyString.isNotEqualTo(
  stringToCheck:= testString1 , 
  unexpected:= testString4 ,
  ignoreCases:= FALSE ,
  message:='' );
  
THIS^.AssertFalse(
	Condition := THIS^.assertorContainer.wasAssertionWrong,
	Message := 'anyStringAssertionTests.isNotEqualTo with stringToCheck:= abcd56ä2&§  , unexpected:= äbcd56ä2&§ , ignoreCases:= False'
);
TEST_FINISHED();


//-------------------------------------------------------------------------------------------------------
TEST('anyStringAssertionTest.isNotEqualTo with stringToCheck:= strangestuff arabic russian , unexpected:= strangestuff arabic russian , ignoreCases:= False ,');

testString5:= "иди сюда кусок дерьма ဒီကိုလာပါ ၊ تعال إلى هنا يا قطعة من الهراء";
testString6:="иди сюда кусок дерьма ဒီကိုလာပါ ၊ تعال إلى هنا يا قطعة من الهراء";

THIS^.assertorContainer.resetAssertor();
THIS^.assertorContainer.assertor.assert.strings.anyString.isNotEqualTo(
  stringToCheck:= testString5 , 
  unexpected:= testString6 ,
  ignoreCases:= FALSE ,
  message:='' );
  
THIS^.AssertTrue(
	Condition := THIS^.assertorContainer.wasAssertionWrong,
	Message := 'anyStringAssertionTests.isNotEqualTo with stringToCheck:= abcd56ä2&§  , unexpected:= äbcd56ä2&§ , ignoreCases:= False'
);
TEST_FINISHED();

//-------------------------------------------------------------------------------------------------------
TEST('anyStringAssertionTest.isNotEqualTo with stringToCheck:= strangestuff arabic russian , unexpected:= strangestuff arabic russian cap, ignoreCases:= False ,');

testString5:= "иди сюда кусок дерьма ဒီကိုလာပါ ၊ تعال إلى هنا يا قطعة من الهراء";
testString6:="иди сюда Кусок дерьма ဒီကိုလာပါ ၊ تعال إلى هنا يا قطعة من الهراء";

THIS^.assertorContainer.resetAssertor();
THIS^.assertorContainer.assertor.assert.strings.anyString.isNotEqualTo(
  stringToCheck:= testString5 , 
  unexpected:= testString6 ,
  ignoreCases:= FALSE ,
  message:='' );
  
THIS^.AssertFalse(
	Condition := THIS^.assertorContainer.wasAssertionWrong,
	Message := 'anyStringAssertionTests.isNotEqualTo with stringToCheck:= abcd56ä2&§  , unexpected:= äbcd56ä2&§ , ignoreCases:= False'
);
TEST_FINISHED();
END_METHOD

(*

short summary
=============

.. <legal notes>

legal notes
=================
| SPDX-FileCopyrightText: © 2023 ekvip automation GmbH <info@ekvip.de>
| SPDX-License-Identifier: Apache-2.0
| For details check: Apache-2.0_

.. _Apache-2.0: https://www.apache.org/licenses/LICENSE-2.0

.. </legal notes>

parameters
==========

*)

{warning 'header is generated please add your documentation'}
METHOD testAnyString_lengthIsExact

VAR
  testString1:STRING(50);
  length: UDINT;
END_VAR
// anyStringAssertionTests.lengthIsExact Tests

//----------------------------------------------------------------------------------------------------------------------------------------
TEST('anyStringAssertionTest.lenghtIsExact with stringToCheck:= EmptyString(50) , expectedLength:= 0');

length := 0;

THIS^.assertorContainer.resetAssertor();
THIS^.assertorContainer.assertor.assert.strings.anyString.lenghtIsExact( 
	stringToCheck	:=	testString1, 
	expectedLength	:=	length,
	message			:=	''             
);

THIS^.AssertFalse(
	Condition	:=	THIS^.assertorContainer.wasAssertionWrong,
	Message		:=	'anyStringAssertionTests.lenghtIsExact with stringToCheck:= EmptyString(50) , expectedLength:= 0'
);

TEST_FINISHED();

//----------------------------------------------------------------------------------------------------------------------------------------

TEST('anyStringAssertionTest.lenghtIsExact with stringToCheck:= Hello World , expectedLength:= 11');

length:= 11;
testString1:= 'Hello World';

THIS^.assertorContainer.resetAssertor();
THIS^.assertorContainer.assertor.assert.strings.anyString.lenghtIsExact( stringToCheck    :=    testString1    , 
                                                       expectedLength   :=    length         ,
                                                       message          :=    ''             ) ;
THIS^.AssertFalse(
	Condition := THIS^.assertorContainer.wasAssertionWrong,
	Message   := 'anyStringAssertionTests.lenghtIsExact with stringToCheck:= Hello World , expectedLength:= 11');

TEST_FINISHED();

//----------------------------------------------------------------------------------------------------------------------------------------

TEST('anyStringAssertionTest.lenghtIsExact with stringToCheck:= Привет, мир , expectedLength:= 11');

length:= 11;
testString1:= 'Привет, мир';

THIS^.assertorContainer.resetAssertor();
THIS^.assertorContainer.assertor.assert.strings.anyString.lenghtIsExact( stringToCheck    :=    testString1    , 
                                                       expectedLength   :=    11             ,
                                                       message          :=    ''             ) ;
THIS^.AssertFalse(
	Condition := THIS^.assertorContainer.wasAssertionWrong,
	Message   := 'anyStringAssertionTests.lenghtIsExact with stringToCheck:= Привет, мир , expectedLength:= 11');

TEST_FINISHED();

//----------------------------------------------------------------------------------------------------------------------------------------

TEST('anyStringAssertionTest.lenghtIsExact with stringToCheck:= 6 spaces , expectedLength:= 6');

length:=6;
testString1:= '      ';

THIS^.assertorContainer.resetAssertor();
THIS^.assertorContainer.assertor.assert.strings.anyString.lenghtIsExact( stringToCheck    :=    testString1    , 
                                                       expectedLength   :=    length         ,
                                                       message          :=    ''             ) ;
THIS^.AssertFalse(
	Condition := THIS^.assertorContainer.wasAssertionWrong,
	Message   := 'anyStringAssertionTests.lenghtIsExact with stringToCheck:= 6 spaces , expectedLength:= 6');

TEST_FINISHED();

//----------------------------------------------------------------------------------------------------------------------------------------

TEST('anyStringAssertionTest.lenghtIsExact with stringToCheck:= Привет, мир Hello , expectedLength:= 17');

length:=17;
testString1:= 'Привет, мир Hello';

THIS^.assertorContainer.resetAssertor();
THIS^.assertorContainer.assertor.assert.strings.anyString.lenghtIsExact( stringToCheck    :=    testString1    , 
                                                       expectedLength   :=    length         ,
                                                       message          :=    ''             ) ;
THIS^.AssertFalse(
	Condition := THIS^.assertorContainer.wasAssertionWrong,
	Message   := 'anyStringAssertionTests.lenghtIsExact with stringToCheck:= Привет, мир Hello , expectedLength:= 17');

TEST_FINISHED();

//----------------------------------------------------------------------------------------------------------------------------------------

TEST('anyStringAssertionTest.lenghtIsExact with stringToCheck:= Привет, мир Hello , expectedLength:= 15');

length:=15;
testString1:= 'Привет, мир Hello';

THIS^.assertorContainer.resetAssertor();
THIS^.assertorContainer.assertor.assert.strings.anyString.lenghtIsExact( stringToCheck    :=    testString1    , 
                                                       expectedLength   :=    length         ,
                                                       message          :=    ''             ) ;
THIS^.AssertTrue(
	Condition := THIS^.assertorContainer.wasAssertionWrong,
	Message   := 'anyStringAssertionTests.lenghtIsExact with stringToCheck:= Привет, мир Hello , expectedLength:= 17');

TEST_FINISHED();
END_METHOD

(*

short summary
=============

.. <legal notes>

legal notes
=================
| SPDX-FileCopyrightText: © 2023 ekvip automation GmbH <info@ekvip.de>
| SPDX-License-Identifier: Apache-2.0
| For details check: Apache-2.0_

.. _Apache-2.0: https://www.apache.org/licenses/LICENSE-2.0

.. </legal notes>

parameters
==========

*)

{warning 'header is generated please add your documentation'}
METHOD testAnyStringContains : BOOL
VAR_INPUT
	inputStruct	: containsDataStr;
	testNumber :USINT;

END_VAR

VAR
	message : STRING;
END_VAR
THIS^.reset();
	

IF (inputStruct.typeToTest = TypeToTest.TEST_WSTRING) THEN
	THIS^.assertorContainer.assertor.assert.strings.anyString.contains(
		stringToCheck 	:= inputStruct.WStringToTest,
		searchString	:= inputStruct.WStringToContain, 
		ignoreCases		:= inputStruct.IgnoreCases,
		message			:= ''
	);			
ELSIF  (inputStruct.typeToTest = TypeToTest.TEST_STRING ) THEN
	THIS^.assertorContainer.assertor.assert.strings.anyString.contains(
		stringToCheck 	:= inputStruct.StringToTest,
		searchString	:= inputStruct.StringToContain, 
		ignoreCases		:= inputStruct.IgnoreCases,
		message			:= ''
	);

END_IF

message	:= CONCAT( 'Test Number ', TO_STRING(testNumber));
message	:= CONCAT( message, ' during function AnyString.contains ');
message	:= CONCAT( Message , ' has failed ');

THIS^.AssertEquals_BOOL(
	Expected 	:= inputStruct.expectedResult,
	Actual 		:= THIS^.assertorContainer.wasAssertionWrong,
	Message 	:= message
);
END_METHOD

(*

short summary
=============

.. <legal notes>

legal notes
=================
| SPDX-FileCopyrightText: © 2023 ekvip automation GmbH <info@ekvip.de>
| SPDX-License-Identifier: Apache-2.0
| For details check: Apache-2.0_

.. _Apache-2.0: https://www.apache.org/licenses/LICENSE-2.0

.. </legal notes>

parameters
==========

*)

{warning 'header is generated please add your documentation'}
METHOD testAnyStringContainsNo : BOOL
VAR_INPUT
	inputStruct	: containsDataStr;
	testNumber 	: USINT;
END_VAR

VAR
	message : STRING;
END_VAR
THIS^.reset();

IF (inputStruct.typeToTest = TypeToTest.TEST_WSTRING) THEN
	THIS^.assertorContainer.assertor.assert.strings.anyString.containsNo(
		stringToCheck 	:= inputStruct.WStringToTest,
		searchString	:= inputStruct.WStringToContain, 
		ignoreCases		:= inputStruct.IgnoreCases,
		message			:= ''
	);
					
ELSIF  (inputStruct.typeToTest = TypeToTest.TEST_STRING ) THEN
	THIS^.assertorContainer.assertor.assert.strings.anyString.containsNo(
		stringToCheck 	:= inputStruct.StringToTest,
		searchString	:= inputStruct.StringToContain, 
		ignoreCases		:= inputStruct.IgnoreCases,
		message			:= ''
	);

END_IF

message	:= CONCAT( 'Test Number ', TO_STRING(testNumber));
message	:= CONCAT( message, ' during function AnyString.containsNo ');
message	:= CONCAT( Message , ' has failed ');

THIS^.AssertEquals_BOOL(
	Expected 	:= inputStruct.expectedResult,
	Actual 		:= THIS^.assertorContainer.wasAssertionWrong,
	Message 	:= message
);
END_METHOD

(*

short summary
=============

.. <legal notes>

legal notes
=================
| SPDX-FileCopyrightText: © 2023 ekvip automation GmbH <info@ekvip.de>
| SPDX-License-Identifier: Apache-2.0
| For details check: Apache-2.0_

.. _Apache-2.0: https://www.apache.org/licenses/LICENSE-2.0

.. </legal notes>

parameters
==========

*)

{warning 'header is generated please add your documentation'}
METHOD testAnyStringEndsWith : BOOL
VAR_INPUT
	inputStruct	: containsDataStr;
	testNumber 	: USINT;
END_VAR

VAR
	message : STRING;
END_VAR
THIS^.reset();

IF (inputStruct.typeToTest = TypeToTest.TEST_WSTRING) THEN
	THIS^.assertorContainer.assertor.assert.strings.anyString.endsWith(
		stringToCheck	:= inputStruct.WStringToTest,
		end				:= inputStruct.WStringToContain,
		ignoreCases		:= inputStruct.IgnoreCases,
		trim			:= inputStruct.Trim,
		message			:= ''
	);
					
ELSIF  (inputStruct.typeToTest = TypeToTest.TEST_STRING ) THEN
	THIS^.assertorContainer.assertor.assert.strings.anyString.endsWith(
		stringToCheck	:= inputStruct.StringToTest,
		end				:= inputStruct.StringToContain,
		ignoreCases		:= inputStruct.IgnoreCases,
		trim			:= inputStruct.Trim,
		message			:= ''
	);
	
END_IF

message	:= CONCAT( 'Test Number ', TO_STRING(testNumber));
message	:= CONCAT( message, ' during function AnyString.endsWith ');
message	:= CONCAT( Message , ' has failed ');

THIS^.AssertEquals_BOOL(
	Expected 	:= inputStruct.expectedResult,
	Actual 		:= THIS^.assertorContainer.wasAssertionWrong,
	Message 	:= message
);
END_METHOD

(*

short summary
=============

.. <legal notes>

legal notes
=================
| SPDX-FileCopyrightText: © 2023 ekvip automation GmbH <info@ekvip.de>
| SPDX-License-Identifier: Apache-2.0
| For details check: Apache-2.0_

.. _Apache-2.0: https://www.apache.org/licenses/LICENSE-2.0

.. </legal notes>

parameters
==========

*)

